KUKA KRL program: EPS_2_26115_SA7003_A_20260219035539.src

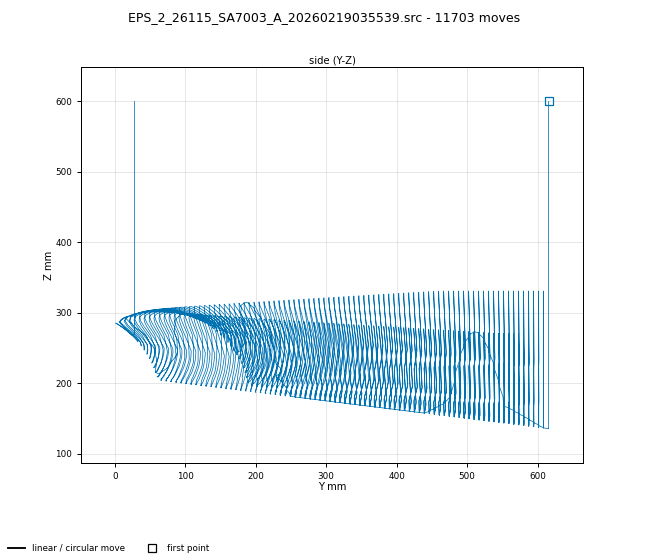
[picture p0: tool path of EPS_2_26115_SA7003_A_20260219035539.src, 11703 of 11705 moves have a stored position in this frame; points joined in program order, loops and branches not executed]
&ACCESS RVP
&REL 4
&COMMENT QRS 19112012
&PARAM EDITMASK = *
DEF PART()
EXT BAS (BAS_COMMAND :IN,REAL :IN )
INT I
BAS (#INITMOV,0 )

;KUKA QRS Post kuka4.cps  Date:22-06-2017 !

File_ID=3058

QRS_PRE_INIT()

;Init var - Until changes are made in qrs_pre_init
Outlet_Square_prg=0
Inlet_1_Square_prg=0
Inlet_2_Square_prg=0
Inlet_3_Square_prg=0
Inlet_4_Square_prg=0
Inlet_5_Square_prg=0

Outlet_1={X 0.000, Y 460.000, Z 230.500, B 0.000, E1 0.000 }
Inlet_1={X 0.000, Y 541.720, Z 170.500, B 0.000, E1 135.000 }
Outlet_1_type=201
Inlet_1_type=201
;QRS#1=Sidecore dimensions
;QRS#2=200-8" PVC SDR 35 Cut Back
;QRS#3=200-8" PVC SDR 35
;QRS#4=
;QRS#5=
;QRS#6=
;QRS#7=
;QRS#8=
;QRS#9=12-08 PSX
;QRS#10=12-08 PSX
;QRS#11=
;QRS#12=
;QRS#13=
;QRS#14=
;QRS#15=
;QRS#16=1220x127x610 2'
;QRS#17=EPS Height
;QRS#18=331
;QRS#19=*
;QRS#20= UPDATED VERSION 22-06-2017
;QRS#21=*
Outlet_Square=0100
Inlet_1_Square=0100
Inlet_2_Square=0
Inlet_3_Square=0
Inlet_4_Square=0
Inlet_5_Square=0
Mill_Square=1
Outlet_Square_Prg=214
Inlet_1_Square_prg=204

QRS_INIT()

$ADVANCE=5

; T1
PTP {E1 173.612,E2 173.612}
PTP {X 0,Y 615.504,A -85,B 0,C 180,E1 173.612,E2 173.612,E3 0,E4 0,E5 0,E6 0}
QRS_SPEED_INIT()
LIN {X 0,Y 615.504,Z 600,A -85,B 0,C 180,E1 173.612,E2 173.612,E3 0,E4 0,E5 0,E6 0} C_VEL
LIN {X 0,Y 615.504,Z 145.874,A -85,B 0,C 180,E1 173.612,E2 173.612} C_VEL
LIN {X 0,Y 615.504,Z 137.7,A -85,B 0,C 180,E1 173.612,E2 173.612} C_VEL
LIN {X 0,Y 615.487,Z 135.7,A -85,B 0,C 180,E1 173.425,E2 173.425} C_VEL
LIN {X 0,Y 615.477,Z 135.7,A -85,B 0,C 180,E1 170.801,E2 170.801} C_VEL
LIN {X 0,Y 615.494,Z 136.005,A -85,B 0,C 180,E1 170.138,E2 170.138} C_VEL
LIN {X 0,Y 615.486,Z 139.365,A -85,B 0,C 180,E1 167.47,E2 167.47} C_VEL
LIN {X 0,Y 615.476,Z 142.627,A -85,B 0,C 180,E1 164.774,E2 164.774} C_VEL
LIN {X 0,Y 615.48,Z 145.054,A -85,B 0,C 180,E1 162.73,E2 162.73} C_VEL
LIN {X 0,Y 615.448,Z 148.65,A -85,B 0,C 180,E1 159.966,E2 159.966} C_VEL
LIN {X 0,Y 615.448,Z 151.726,A -85,B 0,C 180,E1 157.664,E2 157.664} C_VEL
LIN {X 0,Y 615.492,Z 155.32,A -85,B 0,C 180,E1 155.009,E2 155.009} C_VEL
LIN {X 0,Y 615.478,Z 159.371,A -85,B 0,C 180,E1 152.085,E2 152.085} C_VEL
LIN {X 0,Y 615.499,Z 162.507,A -85,B 0,C 180,E1 149.841,E2 149.841} C_VEL
LIN {X 0,Y 615.459,Z 165.766,A -85,B 0,C 180,E1 147.541,E2 147.541} C_VEL
LIN {X 0,Y 615.495,Z 167.197,A -85,B 0,C 180,E1 146.54,E2 146.54} C_VEL
LIN {X 0,Y 615.491,Z 181.195,A -85,B 0,C 180,E1 146.222,E2 146.222} C_VEL
LIN {X 0,Y 615.454,Z 193.523,A -85,B 0,C 180,E1 145.809,E2 145.809} C_VEL
LIN {X 0,Y 615.455,Z 205.838,A -85,B 0,C 180,E1 145.244,E2 145.244} C_VEL
LIN {X 0,Y 615.495,Z 216.991,A -85,B 0,C 180,E1 144.586,E2 144.586} C_VEL
LIN {X 0,Y 615.5,Z 226.768,A -85,B 0,C 180,E1 143.872,E2 143.872} C_VEL
LIN {X 0,Y 615.497,Z 235.818,A -85,B 0,C 180,E1 143.063,E2 143.063} C_VEL
LIN {X 0,Y 615.494,Z 243.879,A -85,B 0,C 180,E1 142.181,E2 142.181} C_VEL
LIN {X 0,Y 615.493,Z 251.897,A -85,B 0,C 180,E1 141.097,E2 141.097} C_VEL
LIN {X 0,Y 615.498,Z 256.903,A -85,B 0,C 180,E1 140.251,E2 140.251} C_VEL
LIN {X 0,Y 615.498,Z 262.112,A -85,B 0,C 180,E1 139.15,E2 139.15} C_VEL
LIN {X 0,Y 615.498,Z 266.306,A -85,B 0,C 180,E1 137.919,E2 137.919} C_VEL
LIN {X 0,Y 615.496,Z 268.876,A -85,B 0,C 180,E1 136.757,E2 136.757} C_VEL
LIN {X 0,Y 615.495,Z 270.003,A -85,B 0,C 180,E1 135.852,E2 135.852} C_VEL
LIN {X 0,Y 615.496,Z 270.387,A -85,B 0,C 180,E1 134.933,E2 134.933} C_VEL
LIN {X 0,Y 615.493,Z 269.961,A -85,B 0,C 180,E1 133.999,E2 133.999} C_VEL
LIN {X 0,Y 615.496,Z 268.703,A -85,B 0,C 180,E1 133.049,E2 133.049} C_VEL
LIN {X 0,Y 615.495,Z 266.55,A -85,B 0,C 180,E1 132.082,E2 132.082} C_VEL
LIN {X 0,Y 615.494,Z 263.4,A -85,B 0,C 180,E1 131.096,E2 131.096} C_VEL
LIN {X 0,Y 615.497,Z 259.108,A -85,B 0,C 180,E1 130.091,E2 130.091} C_VEL
LIN {X 0,Y 615.498,Z 253.468,A -85,B 0,C 180,E1 129.064,E2 129.064} C_VEL
LIN {X 0,Y 615.495,Z 246.196,A -85,B 0,C 180,E1 128.014,E2 128.014} C_VEL
LIN {X 0,Y 615.497,Z 238.191,A -85,B 0,C 180,E1 127.09,E2 127.09} C_VEL
LIN {X 0,Y 615.499,Z 229.604,A -85,B 0,C 180,E1 126.277,E2 126.277} C_VEL
LIN {X 0,Y 615.494,Z 219.814,A -85,B 0,C 180,E1 125.515,E2 125.515} C_VEL
LIN {X 0,Y 615.456,Z 208.685,A -85,B 0,C 180,E1 124.817,E2 124.817} C_VEL
LIN {X 0,Y 615.443,Z 197.705,A -85,B 0,C 180,E1 124.276,E2 124.276} C_VEL
LIN {X 0,Y 615.472,Z 186.221,A -85,B 0,C 180,E1 123.841,E2 123.841} C_VEL
LIN {X 0,Y 615.497,Z 173.65,A -85,B 0,C 180,E1 123.498,E2 123.498} C_VEL
LIN {X 0,Y 615.498,Z 167.193,A -85,B 0,C 180,E1 123.367,E2 123.367} C_VEL
LIN {X 0,Y 615.469,Z 163.712,A -85,B 0,C 180,E1 120.921,E2 120.921} C_VEL
LIN {X 0,Y 615.485,Z 160.236,A -85,B 0,C 180,E1 118.451,E2 118.451} C_VEL
LIN {X 0,Y 615.485,Z 156.237,A -85,B 0,C 180,E1 115.569,E2 115.569} C_VEL
LIN {X 0,Y 615.482,Z 152.529,A -85,B 0,C 180,E1 112.845,E2 112.845} C_VEL
LIN {X 0,Y 615.445,Z 149.456,A -85,B 0,C 180,E1 110.548,E2 110.548} C_VEL
LIN {X 0,Y 615.454,Z 146.046,A -85,B 0,C 180,E1 107.958,E2 107.958} C_VEL
LIN {X 0,Y 615.495,Z 143.494,A -85,B 0,C 180,E1 105.905,E2 105.905} C_VEL
LIN {X 0,Y 615.485,Z 140.188,A -85,B 0,C 180,E1 103.201,E2 103.201} C_VEL
LIN {X 0,Y 615.487,Z 136.889,A -85,B 0,C 180,E1 100.527,E2 100.527} C_VEL
LIN {X 0,Y 615.494,Z 136.061,A -85,B 0,C 180,E1 99.862,E2 99.862} C_VEL
LIN {X 0,Y 615.487,Z 135.702,A -85,B 0,C 180,E1 98.537,E2 98.537} C_VEL
LIN {X 0,Y 615.499,Z 135.696,A -85,B 0,C 180,E1 95.899,E2 95.899} C_VEL
LIN {X 0,Y 615.47,Z 135.7,A -85,B 0,C 180,E1 93.273,E2 93.273} C_VEL
LIN {X 0,Y 615.466,Z 135.7,A -85,B 0,C 180,E1 90.654,E2 90.654} C_VEL
LIN {X 0,Y 615.5,Z 135.693,A -85,B 0,C 180,E1 88.037,E2 88.037} C_VEL
LIN {X 0,Y 615.487,Z 135.699,A -85,B 0,C 180,E1 85.416,E2 85.416} C_VEL
LIN {X 0,Y 615.489,Z 135.702,A -85,B 0,C 180,E1 82.784,E2 82.784} C_VEL
LIN {X 0,Y 615.493,Z 135.697,A -85,B 0,C 180,E1 80.138,E2 80.138} C_VEL
LIN {X 0,Y 615.464,Z 135.701,A -85,B 0,C 180,E1 77.469,E2 77.469} C_VEL
LIN {X 0,Y 615.469,Z 135.7,A -85,B 0,C 180,E1 74.774,E2 74.774} C_VEL
LIN {X 0,Y 615.494,Z 135.699,A -85,B 0,C 180,E1 72.043,E2 72.043} C_VEL
LIN {X 0,Y 615.481,Z 135.699,A -85,B 0,C 180,E1 69.269,E2 69.269} C_VEL
LIN {X 0,Y 615.49,Z 135.695,A -85,B 0,C 180,E1 66.444,E2 66.444} C_VEL
LIN {X 0,Y 615.487,Z 135.701,A -85,B 0,C 180,E1 63.556,E2 63.556} C_VEL
LIN {X 0,Y 615.492,Z 135.695,A -85,B 0,C 180,E1 60.594,E2 60.594} C_VEL
LIN {X 0,Y 615.477,Z 135.7,A -85,B 0,C 180,E1 57.67,E2 57.67} C_VEL
LIN {X 0,Y 615.484,Z 135.7,A -85,B 0,C 180,E1 55.185,E2 55.185} C_VEL
LIN {X 0,Y 615.497,Z 135.697,A -85,B 0,C 180,E1 52.759,E2 52.759} C_VEL
LIN {X 0,Y 615.476,Z 135.7,A -85,B 0,C 180,E1 49.912,E2 49.912} C_VEL
LIN {X 0,Y 615.491,Z 135.695,A -85,B 0,C 180,E1 46.952,E2 46.952} C_VEL
LIN {X 0,Y 615.494,Z 135.701,A -85,B 0,C 180,E1 44.148,E2 44.148} C_VEL
LIN {X 0,Y 615.491,Z 135.694,A -85,B 0,C 180,E1 41.095,E2 41.095} C_VEL
LIN {X 0,Y 615.491,Z 135.701,A -85,B 0,C 180,E1 38.068,E2 38.068} C_VEL
LIN {X 0,Y 615.496,Z 135.699,A -85,B 0,C 180,E1 35.615,E2 35.615} C_VEL
LIN {X 0,Y 615.487,Z 135.702,A -85,B 0,C 180,E1 33.236,E2 33.236} C_VEL
LIN {X 0,Y 615.496,Z 135.7,A -85,B 0,C 180,E1 30.919,E2 30.919} C_VEL
LIN {X 0,Y 615.495,Z 135.701,A -85,B 0,C 180,E1 28.451,E2 28.451} C_VEL
LIN {X 0,Y 615.49,Z 135.695,A -85,B 0,C 180,E1 25.569,E2 25.569} C_VEL
LIN {X 0,Y 615.475,Z 135.699,A -85,B 0,C 180,E1 22.845,E2 22.845} C_VEL
LIN {X 0,Y 615.467,Z 135.7,A -85,B 0,C 180,E1 20.551,E2 20.551} C_VEL
LIN {X 0,Y 615.472,Z 135.7,A -85,B 0,C 180,E1 17.957,E2 17.957} C_VEL
LIN {X 0,Y 615.494,Z 135.7,A -85,B 0,C 180,E1 15.225,E2 15.225} C_VEL
LIN {X 0,Y 615.482,Z 135.699,A -85,B 0,C 180,E1 12.53,E2 12.53} C_VEL
LIN {X 0,Y 615.496,Z 135.693,A -85,B 0,C 180,E1 9.862,E2 9.862} C_VEL
LIN {X 0,Y 615.473,Z 135.699,A -85,B 0,C 180,E1 7.215,E2 7.215} C_VEL
LIN {X 0,Y 615.477,Z 135.7,A -85,B 0,C 180,E1 4.584,E2 4.584} C_VEL
LIN {X 0,Y 615.5,Z 135.699,A -85,B 0,C 180,E1 1.963,E2 1.963} C_VEL
LIN {X 0,Y 615.483,Z 135.701,A -85,B 0,C 180,E1 -0.655,E2 -0.655} C_VEL
LIN {X 0,Y 615.479,Z 135.698,A -85,B 0,C 180,E1 -3.273,E2 -3.273} C_VEL
LIN {X 0,Y 615.498,Z 135.693,A -85,B 0,C 180,E1 -5.899,E2 -5.899} C_VEL
LIN {X 0,Y 615.472,Z 135.699,A -85,B 0,C 180,E1 -8.537,E2 -8.537} C_VEL
LIN {X 0,Y 615.482,Z 135.7,A -85,B 0,C 180,E1 -11.194,E2 -11.194} C_VEL
LIN {X 0,Y 615.486,Z 135.7,A -85,B 0,C 180,E1 -13.932,E2 -13.932} C_VEL
LIN {X 0,Y 615.471,Z 135.7,A -85,B 0,C 180,E1 -16.587,E2 -16.587} C_VEL
LIN {X 0,Y 615.485,Z 135.696,A -85,B 0,C 180,E1 -19.338,E2 -19.338} C_VEL
LIN {X 0,Y 615.49,Z 135.7,A -85,B 0,C 180,E1 -22.137,E2 -22.137} C_VEL
LIN {X 0,Y 615.486,Z 135.697,A -85,B 0,C 180,E1 -24.992,E2 -24.992} C_VEL
LIN {X 0,Y 615.482,Z 135.698,A -85,B 0,C 180,E1 -27.916,E2 -27.916} C_VEL
LIN {X 0,Y 615.465,Z 135.7,A -85,B 0,C 180,E1 -30.162,E2 -30.162} C_VEL
LIN {X 0,Y 615.466,Z 135.7,A -85,B 0,C 180,E1 -32.459,E2 -32.459} C_VEL
LIN {X 0,Y 615.481,Z 135.697,A -85,B 0,C 180,E1 -34.816,E2 -34.816} C_VEL
LIN {X 0,Y 615.494,Z 135.694,A -85,B 0,C 180,E1 -37.242,E2 -37.242} C_VEL
LIN {X 0,Y 615.475,Z 135.7,A -85,B 0,C 180,E1 -40.088,E2 -40.088} C_VEL
LIN {X 0,Y 615.467,Z 135.7,A -85,B 0,C 180,E1 -42.355,E2 -42.355} C_VEL
LIN {X 0,Y 615.497,Z 135.698,A -85,B 0,C 180,E1 -45.068,E2 -45.068} C_VEL
LIN {X 0,Y 615.474,Z 135.7,A -85,B 0,C 180,E1 -47.922,E2 -47.922} C_VEL
LIN {X 0,Y 615.498,Z 135.695,A -85,B 0,C 180,E1 -50.937,E2 -50.937} C_VEL
LIN {X 0,Y 615.487,Z 135.702,A -85,B 0,C 180,E1 -53.575,E2 -53.575} C_VEL
LIN {X 0,Y 615.475,Z 135.817,A -85,B 0,C 180,E1 -54.534,E2 -54.534} C_VEL
LIN {X 0,Y 615.449,Z 144.579,A -85,B 0,C 180,E1 -57.152,E2 -57.152} C_VEL
LIN {X 0,Y 615.438,Z 152.512,A -85,B 0,C 180,E1 -59.458,E2 -59.458} C_VEL
LIN {X 0,Y 615.482,Z 161.755,A -85,B 0,C 180,E1 -62.085,E2 -62.085} C_VEL
LIN {X 0,Y 615.484,Z 171.265,A -85,B 0,C 180,E1 -64.72,E2 -64.72} C_VEL
LIN {X 0,Y 615.471,Z 180.237,A -85,B 0,C 180,E1 -67.155,E2 -67.155} C_VEL
LIN {X 0,Y 615.489,Z 188.8,A -85,B 0,C 180,E1 -69.443,E2 -69.443} C_VEL
LIN {X 0,Y 615.499,Z 200.013,A -85,B 0,C 180,E1 -72.387,E2 -72.387} C_VEL
LIN {X 0,Y 615.48,Z 210.542,A -85,B 0,C 180,E1 -75.113,E2 -75.113} C_VEL
LIN {X 0,Y 615.455,Z 221.087,A -85,B 0,C 180,E1 -77.804,E2 -77.804} C_VEL
LIN {X 0,Y 615.498,Z 223.208,A -85,B 0,C 180,E1 -78.348,E2 -78.348} C_VEL
LIN {X 0,Y 615.497,Z 237.824,A -85,B 0,C 180,E1 -78.64,E2 -78.64} C_VEL
LIN {X 0,Y 615.453,Z 250.972,A -85,B 0,C 180,E1 -79.051,E2 -79.051} C_VEL
LIN {X 0,Y 615.442,Z 262.775,A -85,B 0,C 180,E1 -79.556,E2 -79.556} C_VEL
LIN {X 0,Y 615.489,Z 273.389,A -85,B 0,C 180,E1 -80.138,E2 -80.138} C_VEL
LIN {X 0,Y 615.498,Z 284.233,A -85,B 0,C 180,E1 -80.884,E2 -80.884} C_VEL
LIN {X 0,Y 615.497,Z 294.812,A -85,B 0,C 180,E1 -81.794,E2 -81.794} C_VEL
LIN {X 0,Y 615.498,Z 302.607,A -85,B 0,C 180,E1 -82.62,E2 -82.62} C_VEL
LIN {X 0,Y 615.496,Z 310.203,A -85,B 0,C 180,E1 -83.608,E2 -83.608} C_VEL
LIN {X 0,Y 615.498,Z 317.205,A -85,B 0,C 180,E1 -84.759,E2 -84.759} C_VEL
LIN {X 0,Y 615.494,Z 321.852,A -85,B 0,C 180,E1 -85.744,E2 -85.744} C_VEL
LIN {X 0,Y 615.494,Z 325.399,A -85,B 0,C 180,E1 -86.727,E2 -86.727} C_VEL
LIN {X 0,Y 615.497,Z 327.233,A -85,B 0,C 180,E1 -87.382,E2 -87.382} C_VEL
LIN {X 0,Y 615.5,Z 328.608,A -85,B 0,C 180,E1 -88.037,E2 -88.037} C_VEL
LIN {X 0,Y 615.496,Z 330.174,A -85,B 0,C 180,E1 -89.346,E2 -89.346} C_VEL
LIN {X 0,Y 615.494,Z 330.389,A -85,B 0,C 180,E1 -90,E2 -90} C_VEL
LIN {X 0,Y 615.495,Z 329.58,A -85,B 0,C 180,E1 -91.309,E2 -91.309} C_VEL
LIN {X 0,Y 615.5,Z 328.607,A -85,B 0,C 180,E1 -91.963,E2 -91.963} C_VEL
LIN {X 0,Y 615.497,Z 327.233,A -85,B 0,C 180,E1 -92.618,E2 -92.618} C_VEL
LIN {X 0,Y 615.496,Z 324.349,A -85,B 0,C 180,E1 -93.601,E2 -93.601} C_VEL
LIN {X 0,Y 615.498,Z 320.441,A -85,B 0,C 180,E1 -94.585,E2 -94.585} C_VEL
LIN {X 0,Y 615.499,Z 315.404,A -85,B 0,C 180,E1 -95.57,E2 -95.57} C_VEL
LIN {X 0,Y 615.497,Z 308.87,A -85,B 0,C 180,E1 -96.583,E2 -96.583} C_VEL
LIN {X 0,Y 615.497,Z 301.132,A -85,B 0,C 180,E1 -97.546,E2 -97.546} C_VEL
LIN {X 0,Y 615.498,Z 293.043,A -85,B 0,C 180,E1 -98.371,E2 -98.371} C_VEL
LIN {X 0,Y 615.499,Z 283.165,A -85,B 0,C 180,E1 -99.199,E2 -99.199} C_VEL
LIN {X 0,Y 615.479,Z 271.98,A -85,B 0,C 180,E1 -99.945,E2 -99.945} C_VEL
LIN {X 0,Y 615.441,Z 261.027,A -85,B 0,C 180,E1 -100.528,E2 -100.528} C_VEL
LIN {X 0,Y 615.459,Z 248.774,A -85,B 0,C 180,E1 -101.031,E2 -101.031} C_VEL
LIN {X 0,Y 615.499,Z 236.056,A -85,B 0,C 180,E1 -101.402,E2 -101.402} C_VEL
LIN {X 0,Y 615.498,Z 223.208,A -85,B 0,C 180,E1 -101.652,E2 -101.652} C_VEL
LIN {X 0,Y 615.46,Z 213.08,A -85,B 0,C 180,E1 -104.239,E2 -104.239} C_VEL
LIN {X 0,Y 615.491,Z 202.639,A -85,B 0,C 180,E1 -106.928,E2 -106.928} C_VEL
LIN {X 0,Y 615.487,Z 192.103,A -85,B 0,C 180,E1 -109.685,E2 -109.685} C_VEL
LIN {X 0,Y 615.491,Z 182.087,A -85,B 0,C 180,E1 -112.346,E2 -112.346} C_VEL
LIN {X 0,Y 615.467,Z 172.322,A -85,B 0,C 180,E1 -114.993,E2 -114.993} C_VEL
LIN {X 0,Y 615.496,Z 163.073,A -85,B 0,C 180,E1 -117.545,E2 -117.545} C_VEL
LIN {X 0,Y 615.448,Z 153.832,A -85,B 0,C 180,E1 -120.162,E2 -120.162} C_VEL
LIN {X 0,Y 615.429,Z 145.902,A -85,B 0,C 180,E1 -122.461,E2 -122.461} C_VEL
LIN {X 0,Y 615.496,Z 136.642,A -85,B 0,C 180,E1 -125.214,E2 -125.214} C_VEL
LIN {X 0,Y 615.479,Z 135.7,A -85,B 0,C 180,E1 -125.516,E2 -125.516} C_VEL
LIN {X 0,Y 615.49,Z 135.7,A -85,B 0,C 180,E1 -128.069,E2 -128.069} C_VEL
LIN {X 0,Y 615.49,Z 135.7,A -85,B 0,C 180,E1 -131.094,E2 -131.094} C_VEL
LIN {X 0,Y 615.483,Z 135.7,A -85,B 0,C 180,E1 -133.997,E2 -133.997} C_VEL
LIN {X 0,Y 615.488,Z 135.697,A -85,B 0,C 180,E1 -136.755,E2 -136.755} C_VEL
LIN {X 0,Y 615.485,Z 135.701,A -85,B 0,C 180,E1 -139.393,E2 -139.393} C_VEL
LIN {X 0,Y 615.477,Z 135.701,A -85,B 0,C 180,E1 -141.99,E2 -141.99} C_VEL
LIN {X 0,Y 615.498,Z 135.699,A -85,B 0,C 180,E1 -144.385,E2 -144.385} C_VEL
LIN {X 0,Y 615.492,Z 135.697,A -85,B 0,C 180,E1 -146.764,E2 -146.764} C_VEL
LIN {X 0,Y 615.489,Z 135.698,A -85,B 0,C 180,E1 -149.08,E2 -149.08} C_VEL
LIN {X 0,Y 615.486,Z 135.7,A -85,B 0,C 180,E1 -151.551,E2 -151.551} C_VEL
LIN {X 0,Y 615.499,Z 135.7,A -85,B 0,C 180,E1 -154.43,E2 -154.43} C_VEL
LIN {X 0,Y 615.482,Z 135.7,A -85,B 0,C 180,E1 -157.155,E2 -157.155} C_VEL
LIN {X 0,Y 615.476,Z 135.7,A -85,B 0,C 180,E1 -159.967,E2 -159.967} C_VEL
LIN {X 0,Y 615.484,Z 135.7,A -85,B 0,C 180,E1 -162.729,E2 -162.729} C_VEL
LIN {X 0,Y 615.493,Z 135.7,A -85,B 0,C 180,E1 -165.451,E2 -165.451} C_VEL
LIN {X 0,Y 615.49,Z 135.697,A -85,B 0,C 180,E1 -168.139,E2 -168.139} C_VEL
LIN {X 0,Y 615.484,Z 135.7,A -85,B 0,C 180,E1 -170.801,E2 -170.801} C_VEL
LIN {X 0,Y 615.487,Z 135.7,A -85,B 0,C 180,E1 -173.443,E2 -173.443} C_VEL
LIN {X 0,Y 615.493,Z 135.696,A -85,B 0,C 180,E1 -176.071,E2 -176.071} C_VEL
LIN {X 0,Y 615.495,Z 135.7,A -85,B 0,C 180,E1 -178.691,E2 -178.691} C_VEL
LIN {X 0,Y 615.478,Z 135.7,A -85,B 0,C 180,E1 -181.308,E2 -181.308} C_VEL
LIN {X 0,Y 615.492,Z 135.698,A -85,B 0,C 180,E1 -183.928,E2 -183.928} C_VEL
LIN {X 0,Y 615.487,Z 135.7,A -85,B 0,C 180,E1 -186.575,E2 -186.575} C_VEL
LIN {X 0,Y 614.798,Z 135.845,A -85,B 0,C 180,E1 -187.121,E2 -187.121} C_VEL
LIN {X 0,Y 611.938,Z 136.262,A -85,B 0,C 180,E1 -188.007,E2 -188.007} C_VEL
LIN {X 0,Y 609.539,Z 136.563,A -85,B 0,C 180,E1 -188.719,E2 -188.719} C_VEL
LIN {X 0,Y 608.516,Z 136.702,A -85,B 0,C 180,E1 -189.269,E2 -189.269} C_VEL
LIN {X 0,Y 608.436,Z 136.768,A -85,B 0,C 180,E1 -189.455,E2 -189.455} C_VEL
LIN {X 0,Y 608.462,Z 137.016,A -85,B 0,C 180,E1 -189.977,E2 -189.977} C_VEL
LIN {X 0,Y 608.45,Z 140.401,A -85,B 0,C 180,E1 -192.677,E2 -192.677} C_VEL
LIN {X 0,Y 608.442,Z 143.694,A -85,B 0,C 180,E1 -195.406,E2 -195.406} C_VEL
LIN {X 0,Y 608.442,Z 146.154,A -85,B 0,C 180,E1 -197.476,E2 -197.476} C_VEL
LIN {X 0,Y 608.387,Z 149.724,A -85,B 0,C 180,E1 -200.276,E2 -200.276} C_VEL
LIN {X 0,Y 608.407,Z 153.52,A -85,B 0,C 180,E1 -203.125,E2 -203.125} C_VEL
LIN {X 0,Y 608.413,Z 157.48,A -85,B 0,C 180,E1 -206.037,E2 -206.037} C_VEL
LIN {X 0,Y 608.418,Z 161.039,A -85,B 0,C 180,E1 -208.61,E2 -208.61} C_VEL
LIN {X 0,Y 608.417,Z 164.837,A -85,B 0,C 180,E1 -211.319,E2 -211.319} C_VEL
LIN {X 0,Y 608.427,Z 167.679,A -85,B 0,C 180,E1 -213.325,E2 -213.325} C_VEL
LIN {X 0,Y 608.523,Z 182.01,A -85,B 0,C 180,E1 -213.667,E2 -213.667} C_VEL
LIN {X 0,Y 608.478,Z 193.76,A -85,B 0,C 180,E1 -214.069,E2 -214.069} C_VEL
LIN {X 0,Y 608.455,Z 206.067,A -85,B 0,C 180,E1 -214.64,E2 -214.64} C_VEL
LIN {X 0,Y 608.494,Z 216.768,A -85,B 0,C 180,E1 -215.274,E2 -215.274} C_VEL
LIN {X 0,Y 608.486,Z 227.821,A -85,B 0,C 180,E1 -216.089,E2 -216.089} C_VEL
LIN {X 0,Y 608.46,Z 238.007,A -85,B 0,C 180,E1 -217.036,E2 -217.036} C_VEL
LIN {X 0,Y 608.453,Z 246.33,A -85,B 0,C 180,E1 -217.991,E2 -217.991} C_VEL
LIN {X 0,Y 608.437,Z 254.12,A -85,B 0,C 180,E1 -219.12,E2 -219.12} C_VEL
LIN {X 0,Y 608.452,Z 260.471,A -85,B 0,C 180,E1 -220.303,E2 -220.303} C_VEL
LIN {X 0,Y 608.427,Z 264.671,A -85,B 0,C 180,E1 -221.338,E2 -221.338} C_VEL
LIN {X 0,Y 608.438,Z 267.636,A -85,B 0,C 180,E1 -222.331,E2 -222.331} C_VEL
LIN {X 0,Y 608.433,Z 269.609,A -85,B 0,C 180,E1 -223.305,E2 -223.305} C_VEL
LIN {X 0,Y 608.418,Z 270.697,A -85,B 0,C 180,E1 -224.26,E2 -224.26} C_VEL
LIN {X 0,Y 608.417,Z 270.97,A -85,B 0,C 180,E1 -225.2,E2 -225.2} C_VEL
LIN {X 0,Y 608.427,Z 270.469,A -85,B 0,C 180,E1 -226.126,E2 -226.126} C_VEL
LIN {X 0,Y 608.435,Z 269.189,A -85,B 0,C 180,E1 -227.038,E2 -227.038} C_VEL
LIN {X 0,Y 608.425,Z 267.164,A -85,B 0,C 180,E1 -227.935,E2 -227.935} C_VEL
LIN {X 0,Y 608.431,Z 264.414,A -85,B 0,C 180,E1 -228.821,E2 -228.821} C_VEL
LIN {X 0,Y 608.444,Z 259.863,A -85,B 0,C 180,E1 -229.912,E2 -229.912} C_VEL
LIN {X 0,Y 608.438,Z 253.597,A -85,B 0,C 180,E1 -231.056,E2 -231.056} C_VEL
LIN {X 0,Y 608.453,Z 247.02,A -85,B 0,C 180,E1 -232.008,E2 -232.008} C_VEL
LIN {X 0,Y 608.459,Z 238.894,A -85,B 0,C 180,E1 -232.963,E2 -232.963} C_VEL
LIN {X 0,Y 608.483,Z 228.88,A -85,B 0,C 180,E1 -233.91,E2 -233.91} C_VEL
LIN {X 0,Y 608.486,Z 218.16,A -85,B 0,C 180,E1 -234.725,E2 -234.725} C_VEL
LIN {X 0,Y 608.452,Z 206.176,A -85,B 0,C 180,E1 -235.444,E2 -235.444} C_VEL
LIN {X 0,Y 608.478,Z 194.728,A -85,B 0,C 180,E1 -235.981,E2 -235.981} C_VEL
LIN {X 0,Y 608.523,Z 181.703,A -85,B 0,C 180,E1 -236.432,E2 -236.432} C_VEL
LIN {X 0,Y 608.444,Z 167.665,A -85,B 0,C 180,E1 -236.774,E2 -236.774} C_VEL
LIN {X 0,Y 608.415,Z 163.878,A -85,B 0,C 180,E1 -239.452,E2 -239.452} C_VEL
LIN {X 0,Y 608.43,Z 160.688,A -85,B 0,C 180,E1 -241.732,E2 -241.732} C_VEL
LIN {X 0,Y 608.43,Z 156.596,A -85,B 0,C 180,E1 -244.698,E2 -244.698} C_VEL
LIN {X 0,Y 608.411,Z 152.677,A -85,B 0,C 180,E1 -247.592,E2 -247.592} C_VEL
LIN {X 0,Y 608.42,Z 148.913,A -85,B 0,C 180,E1 -250.428,E2 -250.428} C_VEL
LIN {X 0,Y 608.435,Z 145.048,A -85,B 0,C 180,E1 -253.48,E2 -253.48} C_VEL
LIN {X 0,Y 608.436,Z 142.005,A -85,B 0,C 180,E1 -255.994,E2 -255.994} C_VEL
LIN {X 0,Y 608.451,Z 138.705,A -85,B 0,C 180,E1 -258.676,E2 -258.676} C_VEL
LIN {X 0,Y 608.462,Z 137.049,A -85,B 0,C 180,E1 -260.023,E2 -260.023} C_VEL
LIN {X 0,Y 608.454,Z 136.697,A -85,B 0,C 180,E1 -261.364,E2 -261.364} C_VEL
LIN {X 0,Y 608.491,Z 136.692,A -85,B 0,C 180,E1 -264.033,E2 -264.033} C_VEL
LIN {X 0,Y 608.466,Z 136.693,A -85,B 0,C 180,E1 -266.689,E2 -266.689} C_VEL
LIN {X 0,Y 608.462,Z 136.693,A -85,B 0,C 180,E1 -269.338,E2 -269.338} C_VEL
LIN {X 0,Y 608.469,Z 136.693,A -85,B 0,C 180,E1 -271.986,E2 -271.986} C_VEL
LIN {X 0,Y 608.454,Z 136.696,A -85,B 0,C 180,E1 -274.638,E2 -274.638} C_VEL
LIN {X 0,Y 608.466,Z 136.696,A -85,B 0,C 180,E1 -277.299,E2 -277.299} C_VEL
LIN {X 0,Y 608.46,Z 136.694,A -85,B 0,C 180,E1 -279.977,E2 -279.977} C_VEL
LIN {X 0,Y 608.461,Z 136.693,A -85,B 0,C 180,E1 -282.677,E2 -282.677} C_VEL
LIN {X 0,Y 608.457,Z 136.695,A -85,B 0,C 180,E1 -285.406,E2 -285.406} C_VEL
LIN {X 0,Y 608.447,Z 136.698,A -85,B 0,C 180,E1 -288.172,E2 -288.172} C_VEL
LIN {X 0,Y 608.455,Z 136.694,A -85,B 0,C 180,E1 -290.982,E2 -290.982} C_VEL
LIN {X 0,Y 608.473,Z 136.693,A -85,B 0,C 180,E1 -293.845,E2 -293.845} C_VEL
LIN {X 0,Y 608.447,Z 136.696,A -85,B 0,C 180,E1 -296.774,E2 -296.774} C_VEL
LIN {X 0,Y 608.469,Z 136.693,A -85,B 0,C 180,E1 -299.779,E2 -299.779} C_VEL
LIN {X 0,Y 608.459,Z 136.697,A -85,B 0,C 180,E1 -302.523,E2 -302.523} C_VEL
LIN {X 0,Y 608.436,Z 136.697,A -85,B 0,C 180,E1 -305.278,E2 -305.278} C_VEL
LIN {X 0,Y 608.46,Z 136.694,A -85,B 0,C 180,E1 -307.747,E2 -307.747} C_VEL
LIN {X 0,Y 608.438,Z 136.696,A -85,B 0,C 180,E1 -310.328,E2 -310.328} C_VEL
LIN {X 0,Y 608.458,Z 136.694,A -85,B 0,C 180,E1 -312.959,E2 -312.959} C_VEL
LIN {X 0,Y 608.463,Z 136.696,A -85,B 0,C 180,E1 -315.736,E2 -315.736} C_VEL
LIN {X 0,Y 608.466,Z 136.693,A -85,B 0,C 180,E1 -318.657,E2 -318.657} C_VEL
LIN {X 0,Y 608.469,Z 136.692,A -85,B 0,C 180,E1 -321.413,E2 -321.413} C_VEL
LIN {X 0,Y 608.444,Z 136.696,A -85,B 0,C 180,E1 -323.955,E2 -323.955} C_VEL
LIN {X 0,Y 608.442,Z 136.696,A -85,B 0,C 180,E1 -326.328,E2 -326.328} C_VEL
LIN {X 0,Y 608.48,Z 136.691,A -85,B 0,C 180,E1 -328.727,E2 -328.727} C_VEL
LIN {X 0,Y 608.475,Z 136.694,A -85,B 0,C 180,E1 -331.38,E2 -331.38} C_VEL
LIN {X 0,Y 608.474,Z 136.693,A -85,B 0,C 180,E1 -334.279,E2 -334.279} C_VEL
LIN {X 0,Y 608.446,Z 136.695,A -85,B 0,C 180,E1 -336.876,E2 -336.876} C_VEL
LIN {X 0,Y 608.452,Z 136.694,A -85,B 0,C 180,E1 -339.326,E2 -339.326} C_VEL
LIN {X 0,Y 608.437,Z 136.696,A -85,B 0,C 180,E1 -341.828,E2 -341.828} C_VEL
LIN {X 0,Y 608.477,Z 136.693,A -85,B 0,C 180,E1 -344.595,E2 -344.595} C_VEL
LIN {X 0,Y 608.471,Z 136.695,A -85,B 0,C 180,E1 -347.323,E2 -347.323} C_VEL
LIN {X 0,Y 608.464,Z 136.693,A -85,B 0,C 180,E1 -350.023,E2 -350.023} C_VEL
LIN {X 0,Y 608.441,Z 136.696,A -85,B 0,C 180,E1 -352.701,E2 -352.701} C_VEL
LIN {X 0,Y 608.445,Z 136.696,A -85,B 0,C 180,E1 -355.363,E2 -355.363} C_VEL
LIN {X 0,Y 608.468,Z 136.695,A -85,B 0,C 180,E1 -358.015,E2 -358.015} C_VEL
LIN {X 0,Y 608.477,Z 136.693,A -85,B 0,C 180,E1 -360.662,E2 -360.662} C_VEL
LIN {X 0,Y 608.474,Z 136.692,A -85,B 0,C 180,E1 -363.311,E2 -363.311} C_VEL
LIN {X 0,Y 608.471,Z 136.692,A -85,B 0,C 180,E1 -365.967,E2 -365.967} C_VEL
LIN {X 0,Y 608.446,Z 136.696,A -85,B 0,C 180,E1 -368.636,E2 -368.636} C_VEL
LIN {X 0,Y 608.476,Z 136.695,A -85,B 0,C 180,E1 -371.324,E2 -371.324} C_VEL
LIN {X 0,Y 608.472,Z 136.693,A -85,B 0,C 180,E1 -374.038,E2 -374.038} C_VEL
LIN {X 0,Y 608.439,Z 136.696,A -85,B 0,C 180,E1 -376.785,E2 -376.785} C_VEL
LIN {X 0,Y 608.45,Z 136.696,A -85,B 0,C 180,E1 -379.571,E2 -379.571} C_VEL
LIN {X 0,Y 608.462,Z 136.695,A -85,B 0,C 180,E1 -382.477,E2 -382.477} C_VEL
LIN {X 0,Y 608.454,Z 136.694,A -85,B 0,C 180,E1 -385.301,E2 -385.301} C_VEL
LIN {X 0,Y 608.454,Z 136.694,A -85,B 0,C 180,E1 -387.518,E2 -387.518} C_VEL
LIN {X 0,Y 608.436,Z 136.696,A -85,B 0,C 180,E1 -389.966,E2 -389.966} C_VEL
LIN {X 0,Y 608.446,Z 136.695,A -85,B 0,C 180,E1 -392.52,E2 -392.52} C_VEL
LIN {X 0,Y 608.444,Z 136.697,A -85,B 0,C 180,E1 -395.278,E2 -395.278} C_VEL
LIN {X 0,Y 608.47,Z 136.694,A -85,B 0,C 180,E1 -397.747,E2 -397.747} C_VEL
LIN {X 0,Y 608.447,Z 136.699,A -85,B 0,C 180,E1 -400.328,E2 -400.328} C_VEL
LIN {X 0,Y 608.475,Z 136.691,A -85,B 0,C 180,E1 -403.309,E2 -403.309} C_VEL
LIN {X 0,Y 608.46,Z 136.695,A -85,B 0,C 180,E1 -406.13,E2 -406.13} C_VEL
LIN {X 0,Y 608.454,Z 136.698,A -85,B 0,C 180,E1 -408.823,E2 -408.823} C_VEL
LIN {X 0,Y 608.44,Z 136.698,A -85,B 0,C 180,E1 -411.41,E2 -411.41} C_VEL
LIN {X 0,Y 608.444,Z 136.697,A -85,B 0,C 180,E1 -413.955,E2 -413.955} C_VEL
LIN {X 0,Y 608.468,Z 136.815,A -85,B 0,C 180,E1 -414.369,E2 -414.369} C_VEL
LIN {X 0,Y 608.499,Z 145.917,A -85,B 0,C 180,E1 -417.123,E2 -417.123} C_VEL
LIN {X 0,Y 608.468,Z 153.86,A -85,B 0,C 180,E1 -419.455,E2 -419.455} C_VEL
LIN {X 0,Y 608.495,Z 163.127,A -85,B 0,C 180,E1 -422.111,E2 -422.111} C_VEL
LIN {X 0,Y 608.475,Z 172.395,A -85,B 0,C 180,E1 -424.7,E2 -424.7} C_VEL
LIN {X 0,Y 608.48,Z 182.986,A -85,B 0,C 180,E1 -427.595,E2 -427.595} C_VEL
LIN {X 0,Y 608.459,Z 193.577,A -85,B 0,C 180,E1 -430.43,E2 -430.43} C_VEL
LIN {X 0,Y 608.45,Z 204.168,A -85,B 0,C 180,E1 -433.216,E2 -433.216} C_VEL
LIN {X 0,Y 608.439,Z 214.889,A -85,B 0,C 180,E1 -435.995,E2 -435.995} C_VEL
LIN {X 0,Y 608.438,Z 223.572,A -85,B 0,C 180,E1 -438.222,E2 -438.222} C_VEL
LIN {X 0,Y 608.55,Z 237.098,A -85,B 0,C 180,E1 -438.488,E2 -438.488} C_VEL
LIN {X 0,Y 608.487,Z 249.517,A -85,B 0,C 180,E1 -438.865,E2 -438.865} C_VEL
LIN {X 0,Y 608.467,Z 261.173,A -85,B 0,C 180,E1 -439.35,E2 -439.35} C_VEL
LIN {X 0,Y 608.478,Z 273.58,A -85,B 0,C 180,E1 -440.023,E2 -440.023} C_VEL
LIN {X 0,Y 608.483,Z 284.475,A -85,B 0,C 180,E1 -440.778,E2 -440.778} C_VEL
LIN {X 0,Y 608.475,Z 295.113,A -85,B 0,C 180,E1 -441.699,E2 -441.699} C_VEL
LIN {X 0,Y 608.471,Z 302.961,A -85,B 0,C 180,E1 -442.534,E2 -442.534} C_VEL
LIN {X 0,Y 608.461,Z 310.287,A -85,B 0,C 180,E1 -443.485,E2 -443.485} C_VEL
LIN {X 0,Y 608.451,Z 315.866,A -85,B 0,C 180,E1 -444.366,E2 -444.366} C_VEL
LIN {X 0,Y 608.432,Z 320.95,A -85,B 0,C 180,E1 -445.362,E2 -445.362} C_VEL
LIN {X 0,Y 608.449,Z 324.896,A -85,B 0,C 180,E1 -446.358,E2 -446.358} C_VEL
LIN {X 0,Y 608.425,Z 327.809,A -85,B 0,C 180,E1 -447.352,E2 -447.352} C_VEL
LIN {X 0,Y 608.445,Z 329.201,A -85,B 0,C 180,E1 -448.014,E2 -448.014} C_VEL
LIN {X 0,Y 608.438,Z 330.783,A -85,B 0,C 180,E1 -449.338,E2 -449.338} C_VEL
LIN {X 0,Y 608.434,Z 331,A -85,B 0,C 180,E1 -450,E2 -450} C_VEL
LIN {X 0,Y 608.448,Z 330.184,A -85,B 0,C 180,E1 -451.324,E2 -451.324} C_VEL
LIN {X 0,Y 608.445,Z 329.201,A -85,B 0,C 180,E1 -451.986,E2 -451.986} C_VEL
LIN {X 0,Y 608.425,Z 327.809,A -85,B 0,C 180,E1 -452.648,E2 -452.648} C_VEL
LIN {X 0,Y 608.449,Z 324.896,A -85,B 0,C 180,E1 -453.643,E2 -453.643} C_VEL
LIN {X 0,Y 608.432,Z 320.949,A -85,B 0,C 180,E1 -454.638,E2 -454.638} C_VEL
LIN {X 0,Y 608.438,Z 314.876,A -85,B 0,C 180,E1 -455.801,E2 -455.801} C_VEL
LIN {X 0,Y 608.462,Z 308.234,A -85,B 0,C 180,E1 -456.799,E2 -456.799} C_VEL
LIN {X 0,Y 608.456,Z 299.988,A -85,B 0,C 180,E1 -457.8,E2 -457.8} C_VEL
LIN {X 0,Y 608.472,Z 291.534,A -85,B 0,C 180,E1 -458.636,E2 -458.636} C_VEL
LIN {X 0,Y 608.48,Z 281.088,A -85,B 0,C 180,E1 -459.473,E2 -459.473} C_VEL
LIN {X 0,Y 608.488,Z 270.752,A -85,B 0,C 180,E1 -460.145,E2 -460.145} C_VEL
LIN {X 0,Y 608.466,Z 259.856,A -85,B 0,C 180,E1 -460.713,E2 -460.713} C_VEL
LIN {X 0,Y 608.493,Z 248.085,A -85,B 0,C 180,E1 -461.186,E2 -461.186} C_VEL
LIN {X 0,Y 608.551,Z 235.26,A -85,B 0,C 180,E1 -461.555,E2 -461.555} C_VEL
LIN {X 0,Y 608.442,Z 223.53,A -85,B 0,C 180,E1 -461.789,E2 -461.789} C_VEL
LIN {X 0,Y 608.41,Z 213.435,A -85,B 0,C 180,E1 -464.38,E2 -464.38} C_VEL
LIN {X 0,Y 608.45,Z 204.167,A -85,B 0,C 180,E1 -466.784,E2 -466.784} C_VEL
LIN {X 0,Y 608.46,Z 193.576,A -85,B 0,C 180,E1 -469.571,E2 -469.571} C_VEL
LIN {X 0,Y 608.463,Z 182.724,A -85,B 0,C 180,E1 -472.476,E2 -472.476} C_VEL
LIN {X 0,Y 608.475,Z 172.394,A -85,B 0,C 180,E1 -475.3,E2 -475.3} C_VEL
LIN {X 0,Y 608.495,Z 163.126,A -85,B 0,C 180,E1 -477.89,E2 -477.89} C_VEL
LIN {X 0,Y 608.469,Z 153.859,A -85,B 0,C 180,E1 -480.545,E2 -480.545} C_VEL
LIN {X 0,Y 608.52,Z 144.592,A -85,B 0,C 180,E1 -483.271,E2 -483.271} C_VEL
LIN {X 0,Y 608.471,Z 136.694,A -85,B 0,C 180,E1 -485.682,E2 -485.682} C_VEL
LIN {X 0,Y 608.471,Z 136.696,A -85,B 0,C 180,E1 -488.24,E2 -488.24} C_VEL
LIN {X 0,Y 608.462,Z 136.696,A -85,B 0,C 180,E1 -491.342,E2 -491.342} C_VEL
LIN {X 0,Y 608.462,Z 136.697,A -85,B 0,C 180,E1 -494.264,E2 -494.264} C_VEL
LIN {X 0,Y 608.457,Z 136.696,A -85,B 0,C 180,E1 -497.04,E2 -497.04} C_VEL
LIN {X 0,Y 608.457,Z 136.695,A -85,B 0,C 180,E1 -499.697,E2 -499.697} C_VEL
LIN {X 0,Y 608.467,Z 136.696,A -85,B 0,C 180,E1 -502.253,E2 -502.253} C_VEL
LIN {X 0,Y 608.485,Z 136.692,A -85,B 0,C 180,E1 -505.09,E2 -505.09} C_VEL
LIN {X 0,Y 608.465,Z 136.694,A -85,B 0,C 180,E1 -507.905,E2 -507.905} C_VEL
LIN {X 0,Y 608.47,Z 136.695,A -85,B 0,C 180,E1 -510.22,E2 -510.22} C_VEL
LIN {X 0,Y 608.481,Z 136.692,A -85,B 0,C 180,E1 -512.793,E2 -512.793} C_VEL
LIN {X 0,Y 608.45,Z 136.699,A -85,B 0,C 180,E1 -515.428,E2 -515.428} C_VEL
LIN {X 0,Y 608.47,Z 136.695,A -85,B 0,C 180,E1 -518.308,E2 -518.308} C_VEL
LIN {X 0,Y 608.476,Z 136.694,A -85,B 0,C 180,E1 -521.284,E2 -521.284} C_VEL
LIN {X 0,Y 608.462,Z 136.694,A -85,B 0,C 180,E1 -523.906,E2 -523.906} C_VEL
LIN {X 0,Y 608.462,Z 136.696,A -85,B 0,C 180,E1 -526.643,E2 -526.643} C_VEL
LIN {X 0,Y 608.465,Z 136.695,A -85,B 0,C 180,E1 -529.35,E2 -529.35} C_VEL
LIN {X 0,Y 608.483,Z 136.692,A -85,B 0,C 180,E1 -532.033,E2 -532.033} C_VEL
LIN {X 0,Y 608.469,Z 136.695,A -85,B 0,C 180,E1 -534.698,E2 -534.698} C_VEL
LIN {X 0,Y 608.474,Z 136.693,A -85,B 0,C 180,E1 -537.352,E2 -537.352} C_VEL
LIN {X 0,Y 608.484,Z 136.692,A -85,B 0,C 180,E1 -540,E2 -540} C_VEL
LIN {X 0,Y 608.481,Z 136.694,A -85,B 0,C 180,E1 -542.648,E2 -542.648} C_VEL
LIN {X 0,Y 608.457,Z 136.695,A -85,B 0,C 180,E1 -545.302,E2 -545.302} C_VEL
LIN {X 0,Y 608.481,Z 136.693,A -85,B 0,C 180,E1 -547.967,E2 -547.967} C_VEL
LIN {X 0,Y 608.436,Z 136.768,A -85,B 0,C 180,E1 -549.455,E2 -549.455} C_VEL
LIN {X 0,Y 607.772,Z 137.224,A -85,B 0,C 180,E1 -550.006,E2 -550.006} C_VEL
LIN {X 0,Y 604.904,Z 138.492,A -85,B 0,C 180,E1 -550.895,E2 -550.895} C_VEL
LIN {X 0,Y 602.477,Z 139.614,A -85,B 0,C 180,E1 -551.609,E2 -551.609} C_VEL
LIN {X 0,Y 601.436,Z 140.391,A -85,B 0,C 180,E1 -552.161,E2 -552.161} C_VEL
LIN {X 0,Y 601.353,Z 140.628,A -85,B 0,C 180,E1 -552.349,E2 -552.349} C_VEL
LIN {X 0,Y 601.369,Z 143.712,A -85,B 0,C 180,E1 -554.898,E2 -554.898} C_VEL
LIN {X 0,Y 601.374,Z 147.038,A -85,B 0,C 180,E1 -557.689,E2 -557.689} C_VEL
LIN {X 0,Y 601.329,Z 150.775,A -85,B 0,C 180,E1 -560.772,E2 -560.772} C_VEL
LIN {X 0,Y 601.326,Z 154.266,A -85,B 0,C 180,E1 -563.414,E2 -563.414} C_VEL
LIN {X 0,Y 601.325,Z 157.542,A -85,B 0,C 180,E1 -565.849,E2 -565.849} C_VEL
LIN {X 0,Y 601.327,Z 161.344,A -85,B 0,C 180,E1 -568.632,E2 -568.632} C_VEL
LIN {X 0,Y 601.317,Z 164.55,A -85,B 0,C 180,E1 -570.947,E2 -570.947} C_VEL
LIN {X 0,Y 601.337,Z 167.689,A -85,B 0,C 180,E1 -573.192,E2 -573.192} C_VEL
LIN {X 0,Y 601.608,Z 173.507,A -85,B 0,C 180,E1 -573.314,E2 -573.314} C_VEL
LIN {X 0,Y 601.559,Z 185.9,A -85,B 0,C 180,E1 -573.656,E2 -573.656} C_VEL
LIN {X 0,Y 601.473,Z 197.838,A -85,B 0,C 180,E1 -574.115,E2 -574.115} C_VEL
LIN {X 0,Y 601.475,Z 209.803,A -85,B 0,C 180,E1 -574.724,E2 -574.724} C_VEL
LIN {X 0,Y 601.466,Z 221.496,A -85,B 0,C 180,E1 -575.49,E2 -575.49} C_VEL
LIN {X 0,Y 601.439,Z 231.051,A -85,B 0,C 180,E1 -576.265,E2 -576.265} C_VEL
LIN {X 0,Y 601.415,Z 240.303,A -85,B 0,C 180,E1 -577.188,E2 -577.188} C_VEL
LIN {X 0,Y 601.391,Z 249.001,A -85,B 0,C 180,E1 -578.27,E2 -578.27} C_VEL
LIN {X 0,Y 601.384,Z 255.761,A -85,B 0,C 180,E1 -579.325,E2 -579.325} C_VEL
LIN {X 0,Y 601.336,Z 261.846,A -85,B 0,C 180,E1 -580.564,E2 -580.564} C_VEL
LIN {X 0,Y 601.345,Z 266.197,A -85,B 0,C 180,E1 -581.771,E2 -581.771} C_VEL
LIN {X 0,Y 601.342,Z 268.487,A -85,B 0,C 180,E1 -582.676,E2 -582.676} C_VEL
LIN {X 0,Y 601.343,Z 270.054,A -85,B 0,C 180,E1 -583.593,E2 -583.593} C_VEL
LIN {X 0,Y 601.334,Z 270.881,A -85,B 0,C 180,E1 -584.526,E2 -584.526} C_VEL
LIN {X 0,Y 601.334,Z 270.907,A -85,B 0,C 180,E1 -585.473,E2 -585.473} C_VEL
LIN {X 0,Y 601.343,Z 270.125,A -85,B 0,C 180,E1 -586.435,E2 -586.435} C_VEL
LIN {X 0,Y 601.342,Z 268.483,A -85,B 0,C 180,E1 -587.416,E2 -587.416} C_VEL
LIN {X 0,Y 601.344,Z 265.894,A -85,B 0,C 180,E1 -588.415,E2 -588.415} C_VEL
LIN {X 0,Y 601.332,Z 262.229,A -85,B 0,C 180,E1 -589.435,E2 -589.435} C_VEL
LIN {X 0,Y 601.385,Z 256.255,A -85,B 0,C 180,E1 -590.674,E2 -590.674} C_VEL
LIN {X 0,Y 601.39,Z 249.662,A -85,B 0,C 180,E1 -591.729,E2 -591.729} C_VEL
LIN {X 0,Y 601.415,Z 241.103,A -85,B 0,C 180,E1 -592.811,E2 -592.811} C_VEL
LIN {X 0,Y 601.44,Z 232.07,A -85,B 0,C 180,E1 -593.734,E2 -593.734} C_VEL
LIN {X 0,Y 601.461,Z 221.561,A -85,B 0,C 180,E1 -594.596,E2 -594.596} C_VEL
LIN {X 0,Y 601.456,Z 211.342,A -85,B 0,C 180,E1 -595.274,E2 -595.274} C_VEL
LIN {X 0,Y 601.46,Z 199.875,A -85,B 0,C 180,E1 -595.883,E2 -595.883} C_VEL
LIN {X 0,Y 601.541,Z 188.668,A -85,B 0,C 180,E1 -596.342,E2 -596.342} C_VEL
LIN {X 0,Y 601.59,Z 176.012,A -85,B 0,C 180,E1 -596.718,E2 -596.718} C_VEL
LIN {X 0,Y 601.424,Z 168.706,A -85,B 0,C 180,E1 -596.876,E2 -596.876} C_VEL
LIN {X 0,Y 601.322,Z 167.669,A -85,B 0,C 180,E1 -596.912,E2 -596.912} C_VEL
LIN {X 0,Y 601.342,Z 163.545,A -85,B 0,C 180,E1 -599.865,E2 -599.865} C_VEL
LIN {X 0,Y 601.329,Z 159.39,A -85,B 0,C 180,E1 -602.883,E2 -602.883} C_VEL
LIN {X 0,Y 601.327,Z 155.366,A -85,B 0,C 180,E1 -605.854,E2 -605.854} C_VEL
LIN {X 0,Y 601.304,Z 151.512,A -85,B 0,C 180,E1 -608.757,E2 -608.757} C_VEL
LIN {X 0,Y 601.306,Z 148.405,A -85,B 0,C 180,E1 -611.211,E2 -611.211} C_VEL
LIN {X 0,Y 601.362,Z 145.333,A -85,B 0,C 180,E1 -613.711,E2 -613.711} C_VEL
LIN {X 0,Y 601.347,Z 141.995,A -85,B 0,C 180,E1 -616.482,E2 -616.482} C_VEL
LIN {X 0,Y 601.386,Z 138.626,A -85,B 0,C 180,E1 -619.223,E2 -619.223} C_VEL
LIN {X 0,Y 601.399,Z 137.804,A -85,B 0,C 180,E1 -619.904,E2 -619.904} C_VEL
LIN {X 0,Y 601.44,Z 137.571,A -85,B 0,C 180,E1 -622.615,E2 -622.615} C_VEL
LIN {X 0,Y 601.419,Z 137.573,A -85,B 0,C 180,E1 -625.308,E2 -625.308} C_VEL
LIN {X 0,Y 601.437,Z 137.568,A -85,B 0,C 180,E1 -627.991,E2 -627.991} C_VEL
LIN {X 0,Y 601.437,Z 137.568,A -85,B 0,C 180,E1 -630.669,E2 -630.669} C_VEL
LIN {X 0,Y 601.422,Z 137.571,A -85,B 0,C 180,E1 -633.349,E2 -633.349} C_VEL
LIN {X 0,Y 601.436,Z 137.572,A -85,B 0,C 180,E1 -636.037,E2 -636.037} C_VEL
LIN {X 0,Y 601.41,Z 137.572,A -85,B 0,C 180,E1 -638.738,E2 -638.738} C_VEL
LIN {X 0,Y 601.433,Z 137.569,A -85,B 0,C 180,E1 -641.458,E2 -641.458} C_VEL
LIN {X 0,Y 601.417,Z 137.572,A -85,B 0,C 180,E1 -644.205,E2 -644.205} C_VEL
LIN {X 0,Y 601.429,Z 137.572,A -85,B 0,C 180,E1 -646.986,E2 -646.986} C_VEL
LIN {X 0,Y 601.406,Z 137.572,A -85,B 0,C 180,E1 -649.809,E2 -649.809} C_VEL
LIN {X 0,Y 601.41,Z 137.573,A -85,B 0,C 180,E1 -652.683,E2 -652.683} C_VEL
LIN {X 0,Y 601.395,Z 137.574,A -85,B 0,C 180,E1 -654.879,E2 -654.879} C_VEL
LIN {X 0,Y 601.414,Z 137.573,A -85,B 0,C 180,E1 -657.868,E2 -657.868} C_VEL
LIN {X 0,Y 601.446,Z 137.571,A -85,B 0,C 180,E1 -660.163,E2 -660.163} C_VEL
LIN {X 0,Y 601.428,Z 137.57,A -85,B 0,C 180,E1 -663.313,E2 -663.313} C_VEL
LIN {X 0,Y 601.395,Z 137.577,A -85,B 0,C 180,E1 -666.26,E2 -666.26} C_VEL
LIN {X 0,Y 601.427,Z 137.572,A -85,B 0,C 180,E1 -668.471,E2 -668.471} C_VEL
LIN {X 0,Y 601.412,Z 137.574,A -85,B 0,C 180,E1 -670.875,E2 -670.875} C_VEL
LIN {X 0,Y 601.427,Z 137.572,A -85,B 0,C 180,E1 -673.586,E2 -673.586} C_VEL
LIN {X 0,Y 601.427,Z 137.569,A -85,B 0,C 180,E1 -676.428,E2 -676.428} C_VEL
LIN {X 0,Y 601.414,Z 137.575,A -85,B 0,C 180,E1 -679.427,E2 -679.427} C_VEL
LIN {X 0,Y 601.425,Z 137.572,A -85,B 0,C 180,E1 -681.733,E2 -681.733} C_VEL
LIN {X 0,Y 601.389,Z 137.578,A -85,B 0,C 180,E1 -684.246,E2 -684.246} C_VEL
LIN {X 0,Y 601.414,Z 137.575,A -85,B 0,C 180,E1 -686.686,E2 -686.686} C_VEL
LIN {X 0,Y 601.423,Z 137.573,A -85,B 0,C 180,E1 -689.059,E2 -689.059} C_VEL
LIN {X 0,Y 601.435,Z 137.571,A -85,B 0,C 180,E1 -691.374,E2 -691.374} C_VEL
LIN {X 0,Y 601.411,Z 137.574,A -85,B 0,C 180,E1 -694.133,E2 -694.133} C_VEL
LIN {X 0,Y 601.415,Z 137.573,A -85,B 0,C 180,E1 -696.59,E2 -696.59} C_VEL
LIN {X 0,Y 601.42,Z 137.57,A -85,B 0,C 180,E1 -699.478,E2 -699.478} C_VEL
LIN {X 0,Y 601.398,Z 137.573,A -85,B 0,C 180,E1 -701.608,E2 -701.608} C_VEL
LIN {X 0,Y 601.42,Z 137.571,A -85,B 0,C 180,E1 -704.409,E2 -704.409} C_VEL
LIN {X 0,Y 601.417,Z 137.574,A -85,B 0,C 180,E1 -707.172,E2 -707.172} C_VEL
LIN {X 0,Y 601.438,Z 137.569,A -85,B 0,C 180,E1 -709.905,E2 -709.905} C_VEL
LIN {X 0,Y 601.408,Z 137.572,A -85,B 0,C 180,E1 -712.615,E2 -712.615} C_VEL
LIN {X 0,Y 601.414,Z 137.571,A -85,B 0,C 180,E1 -715.308,E2 -715.308} C_VEL
LIN {X 0,Y 601.436,Z 137.571,A -85,B 0,C 180,E1 -717.991,E2 -717.991} C_VEL
LIN {X 0,Y 601.449,Z 137.569,A -85,B 0,C 180,E1 -720.67,E2 -720.67} C_VEL
LIN {X 0,Y 601.426,Z 137.57,A -85,B 0,C 180,E1 -723.35,E2 -723.35} C_VEL
LIN {X 0,Y 601.423,Z 137.57,A -85,B 0,C 180,E1 -726.037,E2 -726.037} C_VEL
LIN {X 0,Y 601.409,Z 137.573,A -85,B 0,C 180,E1 -728.738,E2 -728.738} C_VEL
LIN {X 0,Y 601.436,Z 137.571,A -85,B 0,C 180,E1 -731.458,E2 -731.458} C_VEL
LIN {X 0,Y 601.418,Z 137.571,A -85,B 0,C 180,E1 -734.206,E2 -734.206} C_VEL
LIN {X 0,Y 601.413,Z 137.571,A -85,B 0,C 180,E1 -736.987,E2 -736.987} C_VEL
LIN {X 0,Y 601.402,Z 137.576,A -85,B 0,C 180,E1 -739.81,E2 -739.81} C_VEL
LIN {X 0,Y 601.413,Z 137.571,A -85,B 0,C 180,E1 -742.683,E2 -742.683} C_VEL
LIN {X 0,Y 601.401,Z 137.574,A -85,B 0,C 180,E1 -744.879,E2 -744.879} C_VEL
LIN {X 0,Y 601.424,Z 137.571,A -85,B 0,C 180,E1 -747.364,E2 -747.364} C_VEL
LIN {X 0,Y 601.403,Z 137.572,A -85,B 0,C 180,E1 -750.144,E2 -750.144} C_VEL
LIN {X 0,Y 601.412,Z 137.572,A -85,B 0,C 180,E1 -752.714,E2 -752.714} C_VEL
LIN {X 0,Y 601.398,Z 137.573,A -85,B 0,C 180,E1 -755.112,E2 -755.112} C_VEL
LIN {X 0,Y 601.439,Z 137.568,A -85,B 0,C 180,E1 -757.419,E2 -757.419} C_VEL
LIN {X 0,Y 601.402,Z 137.573,A -85,B 0,C 180,E1 -759.996,E2 -759.996} C_VEL
LIN {X 0,Y 601.409,Z 137.574,A -85,B 0,C 180,E1 -762.671,E2 -762.671} C_VEL
LIN {X 0,Y 601.401,Z 137.573,A -85,B 0,C 180,E1 -765.48,E2 -765.48} C_VEL
LIN {X 0,Y 601.421,Z 137.57,A -85,B 0,C 180,E1 -768.408,E2 -768.408} C_VEL
LIN {X 0,Y 601.435,Z 137.57,A -85,B 0,C 180,E1 -770.875,E2 -770.875} C_VEL
LIN {X 0,Y 601.404,Z 137.574,A -85,B 0,C 180,E1 -773.417,E2 -773.417} C_VEL
LIN {X 0,Y 601.421,Z 137.686,A -85,B 0,C 180,E1 -774.158,E2 -774.158} C_VEL
LIN {X 0,Y 601.541,Z 143.795,A -85,B 0,C 180,E1 -776.049,E2 -776.049} C_VEL
LIN {X 0,Y 601.518,Z 153.86,A -85,B 0,C 180,E1 -779.064,E2 -779.064} C_VEL
LIN {X 0,Y 601.47,Z 161.803,A -85,B 0,C 180,E1 -781.375,E2 -781.375} C_VEL
LIN {X 0,Y 601.481,Z 171.451,A -85,B 0,C 180,E1 -784.12,E2 -784.12} C_VEL
LIN {X 0,Y 601.464,Z 180.338,A -85,B 0,C 180,E1 -786.592,E2 -786.592} C_VEL
LIN {X 0,Y 601.431,Z 190.929,A -85,B 0,C 180,E1 -789.478,E2 -789.478} C_VEL
LIN {X 0,Y 601.406,Z 201.521,A -85,B 0,C 180,E1 -792.312,E2 -792.312} C_VEL
LIN {X 0,Y 601.367,Z 212.112,A -85,B 0,C 180,E1 -795.102,E2 -795.102} C_VEL
LIN {X 0,Y 601.343,Z 221.379,A -85,B 0,C 180,E1 -797.513,E2 -797.513} C_VEL
LIN {X 0,Y 601.375,Z 223.53,A -85,B 0,C 180,E1 -798.071,E2 -798.071} C_VEL
LIN {X 0,Y 601.619,Z 235.27,A -85,B 0,C 180,E1 -798.311,E2 -798.311} C_VEL
LIN {X 0,Y 601.534,Z 248.348,A -85,B 0,C 180,E1 -798.691,E2 -798.691} C_VEL
LIN {X 0,Y 601.482,Z 259.243,A -85,B 0,C 180,E1 -799.132,E2 -799.132} C_VEL
LIN {X 0,Y 601.478,Z 270.757,A -85,B 0,C 180,E1 -799.736,E2 -799.736} C_VEL
LIN {X 0,Y 601.462,Z 282.253,A -85,B 0,C 180,E1 -800.5,E2 -800.5} C_VEL
LIN {X 0,Y 601.436,Z 291.537,A -85,B 0,C 180,E1 -801.262,E2 -801.262} C_VEL
LIN {X 0,Y 601.4,Z 299.99,A -85,B 0,C 180,E1 -802.108,E2 -802.108} C_VEL
LIN {X 0,Y 601.382,Z 308.236,A -85,B 0,C 180,E1 -803.12,E2 -803.12} C_VEL
LIN {X 0,Y 601.373,Z 314.877,A -85,B 0,C 180,E1 -804.131,E2 -804.131} C_VEL
LIN {X 0,Y 601.336,Z 320.95,A -85,B 0,C 180,E1 -805.307,E2 -805.307} C_VEL
LIN {X 0,Y 601.368,Z 324.896,A -85,B 0,C 180,E1 -806.315,E2 -806.315} C_VEL
LIN {X 0,Y 601.325,Z 327.809,A -85,B 0,C 180,E1 -807.321,E2 -807.321} C_VEL
LIN {X 0,Y 601.343,Z 329.202,A -85,B 0,C 180,E1 -807.991,E2 -807.991} C_VEL
LIN {X 0,Y 601.339,Z 330.784,A -85,B 0,C 180,E1 -809.33,E2 -809.33} C_VEL
LIN {X 0,Y 601.335,Z 331,A -85,B 0,C 180,E1 -810,E2 -810} C_VEL
LIN {X 0,Y 601.347,Z 330.184,A -85,B 0,C 180,E1 -811.339,E2 -811.339} C_VEL
LIN {X 0,Y 601.343,Z 329.201,A -85,B 0,C 180,E1 -812.009,E2 -812.009} C_VEL
LIN {X 0,Y 601.325,Z 327.809,A -85,B 0,C 180,E1 -812.68,E2 -812.68} C_VEL
LIN {X 0,Y 601.368,Z 324.896,A -85,B 0,C 180,E1 -813.685,E2 -813.685} C_VEL
LIN {X 0,Y 601.336,Z 320.949,A -85,B 0,C 180,E1 -814.693,E2 -814.693} C_VEL
LIN {X 0,Y 601.373,Z 314.876,A -85,B 0,C 180,E1 -815.869,E2 -815.869} C_VEL
LIN {X 0,Y 601.382,Z 308.234,A -85,B 0,C 180,E1 -816.88,E2 -816.88} C_VEL
LIN {X 0,Y 601.4,Z 299.988,A -85,B 0,C 180,E1 -817.892,E2 -817.892} C_VEL
LIN {X 0,Y 601.436,Z 291.535,A -85,B 0,C 180,E1 -818.738,E2 -818.738} C_VEL
LIN {X 0,Y 601.449,Z 281.089,A -85,B 0,C 180,E1 -819.585,E2 -819.585} C_VEL
LIN {X 0,Y 601.478,Z 270.753,A -85,B 0,C 180,E1 -820.264,E2 -820.264} C_VEL
LIN {X 0,Y 601.483,Z 259.233,A -85,B 0,C 180,E1 -820.869,E2 -820.869} C_VEL
LIN {X 0,Y 601.527,Z 246.332,A -85,B 0,C 180,E1 -821.375,E2 -821.375} C_VEL
LIN {X 0,Y 601.617,Z 233.431,A -85,B 0,C 180,E1 -821.732,E2 -821.732} C_VEL
LIN {X 0,Y 601.376,Z 223.53,A -85,B 0,C 180,E1 -821.93,E2 -821.93} C_VEL
LIN {X 0,Y 601.372,Z 213.435,A -85,B 0,C 180,E1 -824.552,E2 -824.552} C_VEL
LIN {X 0,Y 601.397,Z 202.844,A -85,B 0,C 180,E1 -827.337,E2 -827.337} C_VEL
LIN {X 0,Y 601.424,Z 192.252,A -85,B 0,C 180,E1 -830.165,E2 -830.165} C_VEL
LIN {X 0,Y 601.433,Z 182.985,A -85,B 0,C 180,E1 -832.682,E2 -832.682} C_VEL
LIN {X 0,Y 601.459,Z 173.718,A -85,B 0,C 180,E1 -835.246,E2 -835.246} C_VEL
LIN {X 0,Y 601.503,Z 164.45,A -85,B 0,C 180,E1 -837.863,E2 -837.863} C_VEL
LIN {X 0,Y 601.483,Z 155.183,A -85,B 0,C 180,E1 -840.549,E2 -840.549} C_VEL
LIN {X 0,Y 601.516,Z 147.837,A -85,B 0,C 180,E1 -842.729,E2 -842.729} C_VEL
LIN {X 0,Y 601.582,Z 139.922,A -85,B 0,C 180,E1 -845.137,E2 -845.137} C_VEL
LIN {X 0,Y 601.423,Z 137.573,A -85,B 0,C 180,E1 -845.932,E2 -845.932} C_VEL
LIN {X 0,Y 601.437,Z 137.57,A -85,B 0,C 180,E1 -848.471,E2 -848.471} C_VEL
LIN {X 0,Y 601.427,Z 137.571,A -85,B 0,C 180,E1 -851.593,E2 -851.593} C_VEL
LIN {X 0,Y 601.43,Z 137.571,A -85,B 0,C 180,E1 -854.535,E2 -854.535} C_VEL
LIN {X 0,Y 601.412,Z 137.574,A -85,B 0,C 180,E1 -857.41,E2 -857.41} C_VEL
LIN {X 0,Y 601.447,Z 137.57,A -85,B 0,C 180,E1 -860.464,E2 -860.464} C_VEL
LIN {X 0,Y 601.408,Z 137.575,A -85,B 0,C 180,E1 -863.417,E2 -863.417} C_VEL
LIN {X 0,Y 601.437,Z 137.57,A -85,B 0,C 180,E1 -866.064,E2 -866.064} C_VEL
LIN {X 0,Y 601.435,Z 137.571,A -85,B 0,C 180,E1 -868.544,E2 -868.544} C_VEL
LIN {X 0,Y 601.435,Z 137.572,A -85,B 0,C 180,E1 -871.373,E2 -871.373} C_VEL
LIN {X 0,Y 601.403,Z 137.575,A -85,B 0,C 180,E1 -873.636,E2 -873.636} C_VEL
LIN {X 0,Y 601.419,Z 137.573,A -85,B 0,C 180,E1 -876.589,E2 -876.589} C_VEL
LIN {X 0,Y 601.432,Z 137.573,A -85,B 0,C 180,E1 -879.478,E2 -879.478} C_VEL
LIN {X 0,Y 601.396,Z 137.575,A -85,B 0,C 180,E1 -882.311,E2 -882.311} C_VEL
LIN {X 0,Y 601.414,Z 137.574,A -85,B 0,C 180,E1 -884.408,E2 -884.408} C_VEL
LIN {X 0,Y 601.42,Z 137.572,A -85,B 0,C 180,E1 -887.172,E2 -887.172} C_VEL
LIN {X 0,Y 601.441,Z 137.569,A -85,B 0,C 180,E1 -889.905,E2 -889.905} C_VEL
LIN {X 0,Y 601.443,Z 137.571,A -85,B 0,C 180,E1 -892.615,E2 -892.615} C_VEL
LIN {X 0,Y 601.422,Z 137.572,A -85,B 0,C 180,E1 -895.308,E2 -895.308} C_VEL
LIN {X 0,Y 601.438,Z 137.57,A -85,B 0,C 180,E1 -897.991,E2 -897.991} C_VEL
LIN {X 0,Y 601.456,Z 137.57,A -85,B 0,C 180,E1 -900.669,E2 -900.669} C_VEL
LIN {X 0,Y 601.423,Z 137.571,A -85,B 0,C 180,E1 -903.349,E2 -903.349} C_VEL
LIN {X 0,Y 601.421,Z 137.572,A -85,B 0,C 180,E1 -906.037,E2 -906.037} C_VEL
LIN {X 0,Y 601.411,Z 137.575,A -85,B 0,C 180,E1 -908.738,E2 -908.738} C_VEL
LIN {X 0,Y 601.399,Z 137.807,A -85,B 0,C 180,E1 -910.095,E2 -910.095} C_VEL
LIN {X 0,Y 601.353,Z 140.628,A -85,B 0,C 180,E1 -912.349,E2 -912.349} C_VEL
LIN {X 0,Y 600.689,Z 141.371,A -85,B 0,C 180,E1 -912.904,E2 -912.904} C_VEL
LIN {X 0,Y 597.831,Z 142.717,A -85,B 0,C 180,E1 -913.803,E2 -913.803} C_VEL
LIN {X 0,Y 595.411,Z 143.801,A -85,B 0,C 180,E1 -914.526,E2 -914.526} C_VEL
LIN {X 0,Y 594.367,Z 144.56,A -85,B 0,C 180,E1 -915.085,E2 -915.085} C_VEL
LIN {X 0,Y 594.28,Z 144.794,A -85,B 0,C 180,E1 -915.274,E2 -915.274} C_VEL
LIN {X 0,Y 594.281,Z 147.927,A -85,B 0,C 180,E1 -917.907,E2 -917.907} C_VEL
LIN {X 0,Y 594.265,Z 151.213,A -85,B 0,C 180,E1 -920.78,E2 -920.78} C_VEL
LIN {X 0,Y 594.223,Z 155.016,A -85,B 0,C 180,E1 -923.711,E2 -923.711} C_VEL
LIN {X 0,Y 594.227,Z 158.05,A -85,B 0,C 180,E1 -925.991,E2 -925.991} C_VEL
LIN {X 0,Y 594.222,Z 161.078,A -85,B 0,C 180,E1 -928.235,E2 -928.235} C_VEL
LIN {X 0,Y 594.23,Z 164.264,A -85,B 0,C 180,E1 -930.568,E2 -930.568} C_VEL
LIN {X 0,Y 594.25,Z 167.685,A -85,B 0,C 180,E1 -933.046,E2 -933.046} C_VEL
LIN {X 0,Y 594.668,Z 172.804,A -85,B 0,C 180,E1 -933.159,E2 -933.159} C_VEL
LIN {X 0,Y 594.594,Z 185.062,A -85,B 0,C 180,E1 -933.493,E2 -933.493} C_VEL
LIN {X 0,Y 594.499,Z 197.477,A -85,B 0,C 180,E1 -933.969,E2 -933.969} C_VEL
LIN {X 0,Y 594.467,Z 209.352,A -85,B 0,C 180,E1 -934.574,E2 -934.574} C_VEL
LIN {X 0,Y 594.46,Z 220.981,A -85,B 0,C 180,E1 -935.338,E2 -935.338} C_VEL
LIN {X 0,Y 594.409,Z 230.767,A -85,B 0,C 180,E1 -936.135,E2 -936.135} C_VEL
LIN {X 0,Y 594.348,Z 238.758,A -85,B 0,C 180,E1 -936.924,E2 -936.924} C_VEL
LIN {X 0,Y 594.298,Z 247.251,A -85,B 0,C 180,E1 -937.947,E2 -937.947} C_VEL
LIN {X 0,Y 594.273,Z 254.435,A -85,B 0,C 180,E1 -939.031,E2 -939.031} C_VEL
LIN {X 0,Y 594.284,Z 260.247,A -85,B 0,C 180,E1 -940.142,E2 -940.142} C_VEL
LIN {X 0,Y 594.234,Z 264.192,A -85,B 0,C 180,E1 -941.117,E2 -941.117} C_VEL
LIN {X 0,Y 594.27,Z 267.926,A -85,B 0,C 180,E1 -942.384,E2 -942.384} C_VEL
LIN {X 0,Y 594.245,Z 269.686,A -85,B 0,C 180,E1 -943.31,E2 -943.31} C_VEL
LIN {X 0,Y 594.23,Z 270.704,A -85,B 0,C 180,E1 -944.25,E2 -944.25} C_VEL
LIN {X 0,Y 594.22,Z 270.97,A -85,B 0,C 180,E1 -945.205,E2 -945.205} C_VEL
LIN {X 0,Y 594.235,Z 270.446,A -85,B 0,C 180,E1 -946.173,E2 -946.173} C_VEL
LIN {X 0,Y 594.247,Z 269.066,A -85,B 0,C 180,E1 -947.16,E2 -947.16} C_VEL
LIN {X 0,Y 594.24,Z 265.68,A -85,B 0,C 180,E1 -948.524,E2 -948.524} C_VEL
LIN {X 0,Y 594.252,Z 262.5,A -85,B 0,C 180,E1 -949.423,E2 -949.423} C_VEL
LIN {X 0,Y 594.293,Z 257.367,A -85,B 0,C 180,E1 -950.532,E2 -950.532} C_VEL
LIN {X 0,Y 594.297,Z 250.535,A -85,B 0,C 180,E1 -951.679,E2 -951.679} C_VEL
LIN {X 0,Y 594.333,Z 243.228,A -85,B 0,C 180,E1 -952.658,E2 -952.658} C_VEL
LIN {X 0,Y 594.412,Z 234.12,A -85,B 0,C 180,E1 -953.64,E2 -953.64} C_VEL
LIN {X 0,Y 594.419,Z 224.419,A -85,B 0,C 180,E1 -954.491,E2 -954.491} C_VEL
LIN {X 0,Y 594.442,Z 214.252,A -85,B 0,C 180,E1 -955.218,E2 -955.218} C_VEL
LIN {X 0,Y 594.458,Z 203.183,A -85,B 0,C 180,E1 -955.85,E2 -955.85} C_VEL
LIN {X 0,Y 594.559,Z 190.606,A -85,B 0,C 180,E1 -956.403,E2 -956.403} C_VEL
LIN {X 0,Y 594.643,Z 177.752,A -85,B 0,C 180,E1 -956.814,E2 -956.814} C_VEL
LIN {X 0,Y 594.473,Z 169.319,A -85,B 0,C 180,E1 -957.005,E2 -957.005} C_VEL
LIN {X 0,Y 594.236,Z 167.666,A -85,B 0,C 180,E1 -957.058,E2 -957.058} C_VEL
LIN {X 0,Y 594.236,Z 164.026,A -85,B 0,C 180,E1 -959.696,E2 -959.696} C_VEL
LIN {X 0,Y 594.259,Z 160.159,A -85,B 0,C 180,E1 -962.533,E2 -962.533} C_VEL
LIN {X 0,Y 594.237,Z 156.051,A -85,B 0,C 180,E1 -965.598,E2 -965.598} C_VEL
LIN {X 0,Y 594.212,Z 152.248,A -85,B 0,C 180,E1 -968.491,E2 -968.491} C_VEL
LIN {X 0,Y 594.254,Z 149.145,A -85,B 0,C 180,E1 -971.106,E2 -971.106} C_VEL
LIN {X 0,Y 594.308,Z 146.158,A -85,B 0,C 180,E1 -973.512,E2 -973.512} C_VEL
LIN {X 0,Y 594.272,Z 142.758,A -85,B 0,C 180,E1 -976.318,E2 -976.318} C_VEL
LIN {X 0,Y 594.311,Z 139.389,A -85,B 0,C 180,E1 -979.093,E2 -979.093} C_VEL
LIN {X 0,Y 594.344,Z 138.571,A -85,B 0,C 180,E1 -979.783,E2 -979.783} C_VEL
LIN {X 0,Y 594.393,Z 138.448,A -85,B 0,C 180,E1 -982.527,E2 -982.527} C_VEL
LIN {X 0,Y 594.388,Z 138.449,A -85,B 0,C 180,E1 -985.252,E2 -985.252} C_VEL
LIN {X 0,Y 594.406,Z 138.444,A -85,B 0,C 180,E1 -987.967,E2 -987.967} C_VEL
LIN {X 0,Y 594.41,Z 138.444,A -85,B 0,C 180,E1 -990.677,E2 -990.677} C_VEL
LIN {X 0,Y 594.374,Z 138.45,A -85,B 0,C 180,E1 -993.389,E2 -993.389} C_VEL
LIN {X 0,Y 594.382,Z 138.45,A -85,B 0,C 180,E1 -996.109,E2 -996.109} C_VEL
LIN {X 0,Y 594.377,Z 138.448,A -85,B 0,C 180,E1 -998.842,E2 -998.842} C_VEL
LIN {X 0,Y 594.392,Z 138.446,A -85,B 0,C 180,E1 -1001.596,E2 -1001.596} C_VEL
LIN {X 0,Y 594.387,Z 138.45,A -85,B 0,C 180,E1 -1004.377,E2 -1004.377} C_VEL
LIN {X 0,Y 594.388,Z 138.447,A -85,B 0,C 180,E1 -1007.193,E2 -1007.193} C_VEL
LIN {X 0,Y 594.376,Z 138.448,A -85,B 0,C 180,E1 -1010.054,E2 -1010.054} C_VEL
LIN {X 0,Y 594.364,Z 138.453,A -85,B 0,C 180,E1 -1012.967,E2 -1012.967} C_VEL
LIN {X 0,Y 594.369,Z 138.451,A -85,B 0,C 180,E1 -1015.193,E2 -1015.193} C_VEL
LIN {X 0,Y 594.383,Z 138.449,A -85,B 0,C 180,E1 -1017.527,E2 -1017.527} C_VEL
LIN {X 0,Y 594.397,Z 138.447,A -85,B 0,C 180,E1 -1020.331,E2 -1020.331} C_VEL
LIN {X 0,Y 594.377,Z 138.448,A -85,B 0,C 180,E1 -1022.95,E2 -1022.95} C_VEL
LIN {X 0,Y 594.348,Z 138.452,A -85,B 0,C 180,E1 -1025.409,E2 -1025.409} C_VEL
LIN {X 0,Y 594.379,Z 138.447,A -85,B 0,C 180,E1 -1027.941,E2 -1027.941} C_VEL
LIN {X 0,Y 594.374,Z 138.45,A -85,B 0,C 180,E1 -1030.822,E2 -1030.822} C_VEL
LIN {X 0,Y 594.366,Z 138.452,A -85,B 0,C 180,E1 -1033.3,E2 -1033.3} C_VEL
LIN {X 0,Y 594.366,Z 138.45,A -85,B 0,C 180,E1 -1036.161,E2 -1036.161} C_VEL
LIN {X 0,Y 594.379,Z 138.449,A -85,B 0,C 180,E1 -1039.178,E2 -1039.178} C_VEL
LIN {X 0,Y 594.389,Z 138.448,A -85,B 0,C 180,E1 -1042.06,E2 -1042.06} C_VEL
LIN {X 0,Y 594.361,Z 138.45,A -85,B 0,C 180,E1 -1044.675,E2 -1044.675} C_VEL
LIN {X 0,Y 594.375,Z 138.448,A -85,B 0,C 180,E1 -1047.089,E2 -1047.089} C_VEL
LIN {X 0,Y 594.37,Z 138.448,A -85,B 0,C 180,E1 -1049.675,E2 -1049.675} C_VEL
LIN {X 0,Y 594.375,Z 138.45,A -85,B 0,C 180,E1 -1052.54,E2 -1052.54} C_VEL
LIN {X 0,Y 594.377,Z 138.448,A -85,B 0,C 180,E1 -1054.807,E2 -1054.807} C_VEL
LIN {X 0,Y 594.364,Z 138.45,A -85,B 0,C 180,E1 -1057.265,E2 -1057.265} C_VEL
LIN {X 0,Y 594.371,Z 138.452,A -85,B 0,C 180,E1 -1059.947,E2 -1059.947} C_VEL
LIN {X 0,Y 594.375,Z 138.448,A -85,B 0,C 180,E1 -1062.807,E2 -1062.807} C_VEL
LIN {X 0,Y 594.389,Z 138.448,A -85,B 0,C 180,E1 -1065.827,E2 -1065.827} C_VEL
LIN {X 0,Y 594.381,Z 138.451,A -85,B 0,C 180,E1 -1068.404,E2 -1068.404} C_VEL
LIN {X 0,Y 594.377,Z 138.448,A -85,B 0,C 180,E1 -1071.158,E2 -1071.158} C_VEL
LIN {X 0,Y 594.376,Z 138.448,A -85,B 0,C 180,E1 -1073.892,E2 -1073.892} C_VEL
LIN {X 0,Y 594.386,Z 138.448,A -85,B 0,C 180,E1 -1076.611,E2 -1076.611} C_VEL
LIN {X 0,Y 594.426,Z 138.445,A -85,B 0,C 180,E1 -1079.323,E2 -1079.323} C_VEL
LIN {X 0,Y 594.406,Z 138.445,A -85,B 0,C 180,E1 -1082.033,E2 -1082.033} C_VEL
LIN {X 0,Y 594.382,Z 138.447,A -85,B 0,C 180,E1 -1084.748,E2 -1084.748} C_VEL
LIN {X 0,Y 594.371,Z 138.449,A -85,B 0,C 180,E1 -1087.474,E2 -1087.474} C_VEL
LIN {X 0,Y 594.393,Z 138.449,A -85,B 0,C 180,E1 -1090.216,E2 -1090.216} C_VEL
LIN {X 0,Y 594.366,Z 138.449,A -85,B 0,C 180,E1 -1092.983,E2 -1092.983} C_VEL
LIN {X 0,Y 594.37,Z 138.449,A -85,B 0,C 180,E1 -1095.781,E2 -1095.781} C_VEL
LIN {X 0,Y 594.387,Z 138.45,A -85,B 0,C 180,E1 -1098.618,E2 -1098.618} C_VEL
LIN {X 0,Y 594.369,Z 138.449,A -85,B 0,C 180,E1 -1101.504,E2 -1101.504} C_VEL
LIN {X 0,Y 594.391,Z 138.448,A -85,B 0,C 180,E1 -1104.446,E2 -1104.446} C_VEL
LIN {X 0,Y 594.387,Z 138.447,A -85,B 0,C 180,E1 -1106.7,E2 -1106.7} C_VEL
LIN {X 0,Y 594.383,Z 138.447,A -85,B 0,C 180,E1 -1108.999,E2 -1108.999} C_VEL
LIN {X 0,Y 594.393,Z 138.447,A -85,B 0,C 180,E1 -1111.645,E2 -1111.645} C_VEL
LIN {X 0,Y 594.378,Z 138.449,A -85,B 0,C 180,E1 -1114.58,E2 -1114.58} C_VEL
LIN {X 0,Y 594.392,Z 138.447,A -85,B 0,C 180,E1 -1117.609,E2 -1117.609} C_VEL
LIN {X 0,Y 594.37,Z 138.45,A -85,B 0,C 180,E1 -1120.567,E2 -1120.567} C_VEL
LIN {X 0,Y 594.368,Z 138.448,A -85,B 0,C 180,E1 -1123.3,E2 -1123.3} C_VEL
LIN {X 0,Y 594.362,Z 138.451,A -85,B 0,C 180,E1 -1126.162,E2 -1126.162} C_VEL
LIN {X 0,Y 594.379,Z 138.448,A -85,B 0,C 180,E1 -1128.536,E2 -1128.536} C_VEL
LIN {X 0,Y 594.38,Z 138.451,A -85,B 0,C 180,E1 -1131.297,E2 -1131.297} C_VEL
LIN {X 0,Y 594.393,Z 138.635,A -85,B 0,C 180,E1 -1133.968,E2 -1133.968} C_VEL
LIN {X 0,Y 594.604,Z 143.269,A -85,B 0,C 180,E1 -1135.435,E2 -1135.435} C_VEL
LIN {X 0,Y 594.545,Z 149.888,A -85,B 0,C 180,E1 -1137.463,E2 -1137.463} C_VEL
LIN {X 0,Y 594.515,Z 157.193,A -85,B 0,C 180,E1 -1139.651,E2 -1139.651} C_VEL
LIN {X 0,Y 594.511,Z 167.099,A -85,B 0,C 180,E1 -1142.546,E2 -1142.546} C_VEL
LIN {X 0,Y 594.464,Z 176.366,A -85,B 0,C 180,E1 -1145.185,E2 -1145.185} C_VEL
LIN {X 0,Y 594.411,Z 186.958,A -85,B 0,C 180,E1 -1148.134,E2 -1148.134} C_VEL
LIN {X 0,Y 594.363,Z 197.746,A -85,B 0,C 180,E1 -1151.077,E2 -1151.077} C_VEL
LIN {X 0,Y 594.312,Z 208.14,A -85,B 0,C 180,E1 -1153.865,E2 -1153.865} C_VEL
LIN {X 0,Y 594.332,Z 218.731,A -85,B 0,C 180,E1 -1156.668,E2 -1156.668} C_VEL
LIN {X 0,Y 594.286,Z 223.53,A -85,B 0,C 180,E1 -1157.926,E2 -1157.926} C_VEL
LIN {X 0,Y 594.67,Z 229.234,A -85,B 0,C 180,E1 -1158.042,E2 -1158.042} C_VEL
LIN {X 0,Y 594.614,Z 242.498,A -85,B 0,C 180,E1 -1158.366,E2 -1158.366} C_VEL
LIN {X 0,Y 594.531,Z 254.644,A -85,B 0,C 180,E1 -1158.801,E2 -1158.801} C_VEL
LIN {X 0,Y 594.475,Z 266.209,A -85,B 0,C 180,E1 -1159.355,E2 -1159.355} C_VEL
LIN {X 0,Y 594.465,Z 277.477,A -85,B 0,C 180,E1 -1160.043,E2 -1160.043} C_VEL
LIN {X 0,Y 594.406,Z 287.648,A -85,B 0,C 180,E1 -1160.815,E2 -1160.815} C_VEL
LIN {X 0,Y 594.372,Z 296.788,A -85,B 0,C 180,E1 -1161.672,E2 -1161.672} C_VEL
LIN {X 0,Y 594.316,Z 305.691,A -85,B 0,C 180,E1 -1162.697,E2 -1162.697} C_VEL
LIN {X 0,Y 594.281,Z 312.17,A -85,B 0,C 180,E1 -1163.615,E2 -1163.615} C_VEL
LIN {X 0,Y 594.289,Z 317.681,A -85,B 0,C 180,E1 -1164.571,E2 -1164.571} C_VEL
LIN {X 0,Y 594.27,Z 322.371,A -85,B 0,C 180,E1 -1165.591,E2 -1165.591} C_VEL
LIN {X 0,Y 594.267,Z 325.956,A -85,B 0,C 180,E1 -1166.61,E2 -1166.61} C_VEL
LIN {X 0,Y 594.226,Z 327.809,A -85,B 0,C 180,E1 -1167.289,E2 -1167.289} C_VEL
LIN {X 0,Y 594.242,Z 329.202,A -85,B 0,C 180,E1 -1167.967,E2 -1167.967} C_VEL
LIN {X 0,Y 594.239,Z 330.784,A -85,B 0,C 180,E1 -1169.322,E2 -1169.322} C_VEL
LIN {X 0,Y 594.236,Z 331,A -85,B 0,C 180,E1 -1170,E2 -1170} C_VEL
LIN {X 0,Y 594.247,Z 330.184,A -85,B 0,C 180,E1 -1171.355,E2 -1171.355} C_VEL
LIN {X 0,Y 594.242,Z 329.202,A -85,B 0,C 180,E1 -1172.033,E2 -1172.033} C_VEL
LIN {X 0,Y 594.226,Z 327.809,A -85,B 0,C 180,E1 -1172.712,E2 -1172.712} C_VEL
LIN {X 0,Y 594.289,Z 324.896,A -85,B 0,C 180,E1 -1173.729,E2 -1173.729} C_VEL
LIN {X 0,Y 594.241,Z 320.949,A -85,B 0,C 180,E1 -1174.749,E2 -1174.749} C_VEL
LIN {X 0,Y 594.305,Z 314.876,A -85,B 0,C 180,E1 -1175.939,E2 -1175.939} C_VEL
LIN {X 0,Y 594.308,Z 308.234,A -85,B 0,C 180,E1 -1176.962,E2 -1176.962} C_VEL
LIN {X 0,Y 594.359,Z 299.988,A -85,B 0,C 180,E1 -1177.987,E2 -1177.987} C_VEL
LIN {X 0,Y 594.382,Z 291.535,A -85,B 0,C 180,E1 -1178.842,E2 -1178.842} C_VEL
LIN {X 0,Y 594.431,Z 281.09,A -85,B 0,C 180,E1 -1179.7,E2 -1179.7} C_VEL
LIN {X 0,Y 594.454,Z 270.754,A -85,B 0,C 180,E1 -1180.387,E2 -1180.387} C_VEL
LIN {X 0,Y 594.501,Z 258.77,A -85,B 0,C 180,E1 -1181.019,E2 -1181.019} C_VEL
LIN {X 0,Y 594.56,Z 246.487,A -85,B 0,C 180,E1 -1181.505,E2 -1181.505} C_VEL
LIN {X 0,Y 594.676,Z 233.431,A -85,B 0,C 180,E1 -1181.871,E2 -1181.871} C_VEL
LIN {X 0,Y 594.457,Z 224.85,A -85,B 0,C 180,E1 -1182.038,E2 -1182.038} C_VEL
LIN {X 0,Y 594.288,Z 223.53,A -85,B 0,C 180,E1 -1182.074,E2 -1182.074} C_VEL
LIN {X 0,Y 594.306,Z 213.435,A -85,B 0,C 180,E1 -1184.729,E2 -1184.729} C_VEL
LIN {X 0,Y 594.339,Z 202.844,A -85,B 0,C 180,E1 -1187.55,E2 -1187.55} C_VEL
LIN {X 0,Y 594.384,Z 192.252,A -85,B 0,C 180,E1 -1190.415,E2 -1190.415} C_VEL
LIN {X 0,Y 594.438,Z 181.661,A -85,B 0,C 180,E1 -1193.333,E2 -1193.333} C_VEL
LIN {X 0,Y 594.489,Z 172.031,A -85,B 0,C 180,E1 -1196.042,E2 -1196.042} C_VEL
LIN {X 0,Y 594.479,Z 163.148,A -85,B 0,C 180,E1 -1198.601,E2 -1198.601} C_VEL
LIN {X 0,Y 594.585,Z 153.859,A -85,B 0,C 180,E1 -1201.338,E2 -1201.338} C_VEL
LIN {X 0,Y 594.611,Z 145.916,A -85,B 0,C 180,E1 -1203.747,E2 -1203.747} C_VEL
LIN {X 0,Y 594.513,Z 139.296,A -85,B 0,C 180,E1 -1205.815,E2 -1205.815} C_VEL
LIN {X 0,Y 594.372,Z 138.452,A -85,B 0,C 180,E1 -1206.138,E2 -1206.138} C_VEL
LIN {X 0,Y 594.383,Z 138.448,A -85,B 0,C 180,E1 -1208.805,E2 -1208.805} C_VEL
LIN {X 0,Y 594.386,Z 138.448,A -85,B 0,C 180,E1 -1211.848,E2 -1211.848} C_VEL
LIN {X 0,Y 594.369,Z 138.45,A -85,B 0,C 180,E1 -1214.809,E2 -1214.809} C_VEL
LIN {X 0,Y 594.37,Z 138.45,A -85,B 0,C 180,E1 -1217.624,E2 -1217.624} C_VEL
LIN {X 0,Y 594.398,Z 138.449,A -85,B 0,C 180,E1 -1220.321,E2 -1220.321} C_VEL
LIN {X 0,Y 594.388,Z 138.448,A -85,B 0,C 180,E1 -1222.913,E2 -1222.913} C_VEL
LIN {X 0,Y 594.387,Z 138.447,A -85,B 0,C 180,E1 -1225.861,E2 -1225.861} C_VEL
LIN {X 0,Y 594.384,Z 138.448,A -85,B 0,C 180,E1 -1228.65,E2 -1228.65} C_VEL
LIN {X 0,Y 594.388,Z 138.448,A -85,B 0,C 180,E1 -1231.042,E2 -1231.042} C_VEL
LIN {X 0,Y 594.389,Z 138.447,A -85,B 0,C 180,E1 -1233.977,E2 -1233.977} C_VEL
LIN {X 0,Y 594.388,Z 138.449,A -85,B 0,C 180,E1 -1236.296,E2 -1236.296} C_VEL
LIN {X 0,Y 594.407,Z 138.446,A -85,B 0,C 180,E1 -1239.224,E2 -1239.224} C_VEL
LIN {X 0,Y 594.354,Z 138.451,A -85,B 0,C 180,E1 -1242.095,E2 -1242.095} C_VEL
LIN {X 0,Y 594.368,Z 138.45,A -85,B 0,C 180,E1 -1244.219,E2 -1244.219} C_VEL
LIN {X 0,Y 594.385,Z 138.449,A -85,B 0,C 180,E1 -1246.321,E2 -1246.321} C_VEL
LIN {X 0,Y 594.378,Z 138.449,A -85,B 0,C 180,E1 -1249.094,E2 -1249.094} C_VEL
LIN {X 0,Y 594.418,Z 138.444,A -85,B 0,C 180,E1 -1251.843,E2 -1251.843} C_VEL
LIN {X 0,Y 594.398,Z 138.449,A -85,B 0,C 180,E1 -1254.572,E2 -1254.572} C_VEL
LIN {X 0,Y 594.407,Z 138.445,A -85,B 0,C 180,E1 -1257.289,E2 -1257.289} C_VEL
LIN {X 0,Y 594.42,Z 138.444,A -85,B 0,C 180,E1 -1260,E2 -1260} C_VEL
LIN {X 0,Y 594.411,Z 138.447,A -85,B 0,C 180,E1 -1262.71,E2 -1262.71} C_VEL
LIN {X 0,Y 594.389,Z 138.448,A -85,B 0,C 180,E1 -1265.427,E2 -1265.427} C_VEL
LIN {X 0,Y 594.416,Z 138.444,A -85,B 0,C 180,E1 -1268.156,E2 -1268.156} C_VEL
LIN {X 0,Y 594.345,Z 138.629,A -85,B 0,C 180,E1 -1270.216,E2 -1270.216} C_VEL
LIN {X 0,Y 594.294,Z 142.047,A -85,B 0,C 180,E1 -1272.984,E2 -1272.984} C_VEL
LIN {X 0,Y 594.28,Z 144.794,A -85,B 0,C 180,E1 -1275.274,E2 -1275.274} C_VEL
LIN {X 0,Y 593.605,Z 145.527,A -85,B 0,C 180,E1 -1275.836,E2 -1275.836} C_VEL
LIN {X 0,Y 590.739,Z 146.859,A -85,B 0,C 180,E1 -1276.745,E2 -1276.745} C_VEL
LIN {X 0,Y 588.316,Z 147.939,A -85,B 0,C 180,E1 -1277.476,E2 -1277.476} C_VEL
LIN {X 0,Y 587.27,Z 148.702,A -85,B 0,C 180,E1 -1278.041,E2 -1278.041} C_VEL
LIN {X 0,Y 587.181,Z 148.939,A -85,B 0,C 180,E1 -1278.232,E2 -1278.232} C_VEL
LIN {X 0,Y 587.165,Z 152.222,A -85,B 0,C 180,E1 -1281.043,E2 -1281.043} C_VEL
LIN {X 0,Y 587.112,Z 154.792,A -85,B 0,C 180,E1 -1283.267,E2 -1283.267} C_VEL
LIN {X 0,Y 587.136,Z 157.752,A -85,B 0,C 180,E1 -1285.525,E2 -1285.525} C_VEL
LIN {X 0,Y 587.152,Z 160.812,A -85,B 0,C 180,E1 -1287.827,E2 -1287.827} C_VEL
LIN {X 0,Y 587.155,Z 164.386,A -85,B 0,C 180,E1 -1290.479,E2 -1290.479} C_VEL
LIN {X 0,Y 587.148,Z 167.681,A -85,B 0,C 180,E1 -1292.896,E2 -1292.896} C_VEL
LIN {X 0,Y 587.73,Z 173.634,A -85,B 0,C 180,E1 -1293.036,E2 -1293.036} C_VEL
LIN {X 0,Y 587.63,Z 187.272,A -85,B 0,C 180,E1 -1293.429,E2 -1293.429} C_VEL
LIN {X 0,Y 587.541,Z 198.85,A -85,B 0,C 180,E1 -1293.897,E2 -1293.897} C_VEL
LIN {X 0,Y 587.463,Z 209.654,A -85,B 0,C 180,E1 -1294.466,E2 -1294.466} C_VEL
LIN {X 0,Y 587.439,Z 221.044,A -85,B 0,C 180,E1 -1295.225,E2 -1295.225} C_VEL
LIN {X 0,Y 587.354,Z 231.654,A -85,B 0,C 180,E1 -1296.107,E2 -1296.107} C_VEL
LIN {X 0,Y 587.296,Z 240.012,A -85,B 0,C 180,E1 -1296.964,E2 -1296.964} C_VEL
LIN {X 0,Y 587.22,Z 247.893,A -85,B 0,C 180,E1 -1297.951,E2 -1297.951} C_VEL
LIN {X 0,Y 587.208,Z 255.398,A -85,B 0,C 180,E1 -1299.123,E2 -1299.123} C_VEL
LIN {X 0,Y 587.2,Z 261.049,A -85,B 0,C 180,E1 -1300.263,E2 -1300.263} C_VEL
LIN {X 0,Y 587.141,Z 264.564,A -85,B 0,C 180,E1 -1301.173,E2 -1301.173} C_VEL
LIN {X 0,Y 587.19,Z 267.273,A -85,B 0,C 180,E1 -1302.092,E2 -1302.092} C_VEL
LIN {X 0,Y 587.147,Z 269.384,A -85,B 0,C 180,E1 -1303.1,E2 -1303.1} C_VEL
LIN {X 0,Y 587.155,Z 270.604,A -85,B 0,C 180,E1 -1304.096,E2 -1304.096} C_VEL
LIN {X 0,Y 587.143,Z 270.999,A -85,B 0,C 180,E1 -1305.071,E2 -1305.071} C_VEL
LIN {X 0,Y 587.135,Z 270.578,A -85,B 0,C 180,E1 -1306.031,E2 -1306.031} C_VEL
LIN {X 0,Y 587.163,Z 269.4,A -85,B 0,C 180,E1 -1306.979,E2 -1306.979} C_VEL
LIN {X 0,Y 587.165,Z 266.28,A -85,B 0,C 180,E1 -1308.371,E2 -1308.371} C_VEL
LIN {X 0,Y 587.161,Z 263.034,A -85,B 0,C 180,E1 -1309.342,E2 -1309.342} C_VEL
LIN {X 0,Y 587.208,Z 258.815,A -85,B 0,C 180,E1 -1310.313,E2 -1310.313} C_VEL
LIN {X 0,Y 587.232,Z 253.483,A -85,B 0,C 180,E1 -1311.294,E2 -1311.294} C_VEL
LIN {X 0,Y 587.241,Z 246.102,A -85,B 0,C 180,E1 -1312.384,E2 -1312.384} C_VEL
LIN {X 0,Y 587.277,Z 238.416,A -85,B 0,C 180,E1 -1313.301,E2 -1313.301} C_VEL
LIN {X 0,Y 587.374,Z 229.157,A -85,B 0,C 180,E1 -1314.207,E2 -1314.207} C_VEL
LIN {X 0,Y 587.428,Z 218.605,A -85,B 0,C 180,E1 -1315.045,E2 -1315.045} C_VEL
LIN {X 0,Y 587.473,Z 206.773,A -85,B 0,C 180,E1 -1315.787,E2 -1315.787} C_VEL
LIN {X 0,Y 587.545,Z 195.077,A -85,B 0,C 180,E1 -1316.36,E2 -1316.36} C_VEL
LIN {X 0,Y 587.672,Z 182.245,A -85,B 0,C 180,E1 -1316.826,E2 -1316.826} C_VEL
LIN {X 0,Y 587.512,Z 170.309,A -85,B 0,C 180,E1 -1317.13,E2 -1317.13} C_VEL
LIN {X 0,Y 587.145,Z 167.672,A -85,B 0,C 180,E1 -1317.201,E2 -1317.201} C_VEL
LIN {X 0,Y 587.153,Z 164.103,A -85,B 0,C 180,E1 -1319.819,E2 -1319.819} C_VEL
LIN {X 0,Y 587.163,Z 160.707,A -85,B 0,C 180,E1 -1322.341,E2 -1322.341} C_VEL
LIN {X 0,Y 587.158,Z 156.87,A -85,B 0,C 180,E1 -1325.233,E2 -1325.233} C_VEL
LIN {X 0,Y 587.128,Z 153.068,A -85,B 0,C 180,E1 -1328.218,E2 -1328.218} C_VEL
LIN {X 0,Y 587.188,Z 149.641,A -85,B 0,C 180,E1 -1331.146,E2 -1331.146} C_VEL
LIN {X 0,Y 587.222,Z 146.127,A -85,B 0,C 180,E1 -1334.022,E2 -1334.022} C_VEL
LIN {X 0,Y 587.213,Z 143.568,A -85,B 0,C 180,E1 -1336.151,E2 -1336.151} C_VEL
LIN {X 0,Y 587.266,Z 140.196,A -85,B 0,C 180,E1 -1338.961,E2 -1338.961} C_VEL
LIN {X 0,Y 587.273,Z 139.35,A -85,B 0,C 180,E1 -1339.659,E2 -1339.659} C_VEL
LIN {X 0,Y 587.366,Z 139.322,A -85,B 0,C 180,E1 -1342.437,E2 -1342.437} C_VEL
LIN {X 0,Y 587.359,Z 139.325,A -85,B 0,C 180,E1 -1345.195,E2 -1345.195} C_VEL
LIN {X 0,Y 587.375,Z 139.32,A -85,B 0,C 180,E1 -1347.943,E2 -1347.943} C_VEL
LIN {X 0,Y 587.382,Z 139.319,A -85,B 0,C 180,E1 -1350.685,E2 -1350.685} C_VEL
LIN {X 0,Y 587.326,Z 139.328,A -85,B 0,C 180,E1 -1353.43,E2 -1353.43} C_VEL
LIN {X 0,Y 587.357,Z 139.322,A -85,B 0,C 180,E1 -1355.493,E2 -1355.493} C_VEL
LIN {X 0,Y 587.365,Z 139.323,A -85,B 0,C 180,E1 -1358.255,E2 -1358.255} C_VEL
LIN {X 0,Y 587.345,Z 139.325,A -85,B 0,C 180,E1 -1361.134,E2 -1361.134} C_VEL
LIN {X 0,Y 587.363,Z 139.323,A -85,B 0,C 180,E1 -1364.261,E2 -1364.261} C_VEL
LIN {X 0,Y 587.355,Z 139.322,A -85,B 0,C 180,E1 -1367.406,E2 -1367.406} C_VEL
LIN {X 0,Y 587.331,Z 139.327,A -85,B 0,C 180,E1 -1370.305,E2 -1370.305} C_VEL
LIN {X 0,Y 587.323,Z 139.327,A -85,B 0,C 180,E1 -1373.259,E2 -1373.259} C_VEL
LIN {X 0,Y 587.329,Z 139.327,A -85,B 0,C 180,E1 -1375.517,E2 -1375.517} C_VEL
LIN {X 0,Y 587.345,Z 139.326,A -85,B 0,C 180,E1 -1377.818,E2 -1377.818} C_VEL
LIN {X 0,Y 587.343,Z 139.324,A -85,B 0,C 180,E1 -1380.512,E2 -1380.512} C_VEL
LIN {X 0,Y 587.334,Z 139.326,A -85,B 0,C 180,E1 -1383.397,E2 -1383.397} C_VEL
LIN {X 0,Y 587.289,Z 139.332,A -85,B 0,C 180,E1 -1385.9,E2 -1385.9} C_VEL
LIN {X 0,Y 587.329,Z 139.328,A -85,B 0,C 180,E1 -1388.479,E2 -1388.479} C_VEL
LIN {X 0,Y 587.334,Z 139.327,A -85,B 0,C 180,E1 -1391.157,E2 -1391.157} C_VEL
LIN {X 0,Y 587.324,Z 139.326,A -85,B 0,C 180,E1 -1394.114,E2 -1394.114} C_VEL
LIN {X 0,Y 587.311,Z 139.331,A -85,B 0,C 180,E1 -1396.994,E2 -1396.994} C_VEL
LIN {X 0,Y 587.312,Z 139.329,A -85,B 0,C 180,E1 -1399.746,E2 -1399.746} C_VEL
LIN {X 0,Y 587.346,Z 139.323,A -85,B 0,C 180,E1 -1402.393,E2 -1402.393} C_VEL
LIN {X 0,Y 587.334,Z 139.325,A -85,B 0,C 180,E1 -1404.945,E2 -1404.945} C_VEL
LIN {X 0,Y 587.336,Z 139.325,A -85,B 0,C 180,E1 -1407.421,E2 -1407.421} C_VEL
LIN {X 0,Y 587.319,Z 139.327,A -85,B 0,C 180,E1 -1409.829,E2 -1409.829} C_VEL
LIN {X 0,Y 587.351,Z 139.323,A -85,B 0,C 180,E1 -1412.307,E2 -1412.307} C_VEL
LIN {X 0,Y 587.352,Z 139.325,A -85,B 0,C 180,E1 -1415.242,E2 -1415.242} C_VEL
LIN {X 0,Y 587.325,Z 139.326,A -85,B 0,C 180,E1 -1418.226,E2 -1418.226} C_VEL
LIN {X 0,Y 587.347,Z 139.327,A -85,B 0,C 180,E1 -1421.152,E2 -1421.152} C_VEL
LIN {X 0,Y 587.326,Z 139.326,A -85,B 0,C 180,E1 -1424.025,E2 -1424.025} C_VEL
LIN {X 0,Y 587.317,Z 139.328,A -85,B 0,C 180,E1 -1426.859,E2 -1426.859} C_VEL
LIN {X 0,Y 587.343,Z 139.327,A -85,B 0,C 180,E1 -1429.661,E2 -1429.661} C_VEL
LIN {X 0,Y 587.349,Z 139.324,A -85,B 0,C 180,E1 -1432.437,E2 -1432.437} C_VEL
LIN {X 0,Y 587.356,Z 139.322,A -85,B 0,C 180,E1 -1435.196,E2 -1435.196} C_VEL
LIN {X 0,Y 587.374,Z 139.322,A -85,B 0,C 180,E1 -1437.943,E2 -1437.943} C_VEL
LIN {X 0,Y 587.391,Z 139.32,A -85,B 0,C 180,E1 -1440.686,E2 -1440.686} C_VEL
LIN {X 0,Y 587.33,Z 139.326,A -85,B 0,C 180,E1 -1443.43,E2 -1443.43} C_VEL
LIN {X 0,Y 587.332,Z 139.326,A -85,B 0,C 180,E1 -1446.183,E2 -1446.183} C_VEL
LIN {X 0,Y 587.327,Z 139.329,A -85,B 0,C 180,E1 -1448.95,E2 -1448.95} C_VEL
LIN {X 0,Y 587.344,Z 139.324,A -85,B 0,C 180,E1 -1451.737,E2 -1451.737} C_VEL
LIN {X 0,Y 587.336,Z 139.325,A -85,B 0,C 180,E1 -1454.554,E2 -1454.554} C_VEL
LIN {X 0,Y 587.345,Z 139.327,A -85,B 0,C 180,E1 -1457.406,E2 -1457.406} C_VEL
LIN {X 0,Y 587.314,Z 139.329,A -85,B 0,C 180,E1 -1459.576,E2 -1459.576} C_VEL
LIN {X 0,Y 587.34,Z 139.325,A -85,B 0,C 180,E1 -1462.514,E2 -1462.514} C_VEL
LIN {X 0,Y 587.337,Z 139.325,A -85,B 0,C 180,E1 -1465.517,E2 -1465.517} C_VEL
LIN {X 0,Y 587.35,Z 139.323,A -85,B 0,C 180,E1 -1467.818,E2 -1467.818} C_VEL
LIN {X 0,Y 587.329,Z 139.327,A -85,B 0,C 180,E1 -1470.508,E2 -1470.508} C_VEL
LIN {X 0,Y 587.337,Z 139.328,A -85,B 0,C 180,E1 -1473.111,E2 -1473.111} C_VEL
LIN {X 0,Y 587.293,Z 139.33,A -85,B 0,C 180,E1 -1475.9,E2 -1475.9} C_VEL
LIN {X 0,Y 587.325,Z 139.326,A -85,B 0,C 180,E1 -1478.48,E2 -1478.48} C_VEL
LIN {X 0,Y 587.339,Z 139.325,A -85,B 0,C 180,E1 -1481.157,E2 -1481.157} C_VEL
LIN {X 0,Y 587.33,Z 139.327,A -85,B 0,C 180,E1 -1484.114,E2 -1484.114} C_VEL
LIN {X 0,Y 587.319,Z 139.326,A -85,B 0,C 180,E1 -1486.994,E2 -1486.994} C_VEL
LIN {X 0,Y 587.319,Z 139.328,A -85,B 0,C 180,E1 -1489.746,E2 -1489.746} C_VEL
LIN {X 0,Y 587.345,Z 139.327,A -85,B 0,C 180,E1 -1492.392,E2 -1492.392} C_VEL
LIN {X 0,Y 587.347,Z 139.463,A -85,B 0,C 180,E1 -1493.733,E2 -1493.733} C_VEL
LIN {X 0,Y 587.662,Z 143.269,A -85,B 0,C 180,E1 -1494.967,E2 -1494.967} C_VEL
LIN {X 0,Y 587.653,Z 149.27,A -85,B 0,C 180,E1 -1496.842,E2 -1496.842} C_VEL
LIN {X 0,Y 587.545,Z 157.871,A -85,B 0,C 180,E1 -1499.456,E2 -1499.456} C_VEL
LIN {X 0,Y 587.53,Z 167.383,A -85,B 0,C 180,E1 -1502.275,E2 -1502.275} C_VEL
LIN {X 0,Y 587.451,Z 177.69,A -85,B 0,C 180,E1 -1505.246,E2 -1505.246} C_VEL
LIN {X 0,Y 587.388,Z 188.282,A -85,B 0,C 180,E1 -1508.228,E2 -1508.228} C_VEL
LIN {X 0,Y 587.313,Z 198.873,A -85,B 0,C 180,E1 -1511.15,E2 -1511.15} C_VEL
LIN {X 0,Y 587.257,Z 209.464,A -85,B 0,C 180,E1 -1514.023,E2 -1514.023} C_VEL
LIN {X 0,Y 587.234,Z 220.055,A -85,B 0,C 180,E1 -1516.857,E2 -1516.857} C_VEL
LIN {X 0,Y 587.198,Z 223.572,A -85,B 0,C 180,E1 -1517.789,E2 -1517.789} C_VEL
LIN {X 0,Y 587.74,Z 228.092,A -85,B 0,C 180,E1 -1517.877,E2 -1517.877} C_VEL
LIN {X 0,Y 587.672,Z 241.739,A -85,B 0,C 180,E1 -1518.204,E2 -1518.204} C_VEL
LIN {X 0,Y 587.564,Z 254.425,A -85,B 0,C 180,E1 -1518.657,E2 -1518.657} C_VEL
LIN {X 0,Y 587.477,Z 266.21,A -85,B 0,C 180,E1 -1519.227,E2 -1519.227} C_VEL
LIN {X 0,Y 587.462,Z 277.477,A -85,B 0,C 180,E1 -1519.924,E2 -1519.924} C_VEL
LIN {X 0,Y 587.384,Z 287.648,A -85,B 0,C 180,E1 -1520.705,E2 -1520.705} C_VEL
LIN {X 0,Y 587.34,Z 296.788,A -85,B 0,C 180,E1 -1521.571,E2 -1521.571} C_VEL
LIN {X 0,Y 587.259,Z 305.692,A -85,B 0,C 180,E1 -1522.608,E2 -1522.608} C_VEL
LIN {X 0,Y 587.195,Z 312.747,A -85,B 0,C 180,E1 -1523.627,E2 -1523.627} C_VEL
LIN {X 0,Y 587.211,Z 317.681,A -85,B 0,C 180,E1 -1524.506,E2 -1524.506} C_VEL
LIN {X 0,Y 587.188,Z 322.372,A -85,B 0,C 180,E1 -1525.538,E2 -1525.538} C_VEL
LIN {X 0,Y 587.193,Z 325.956,A -85,B 0,C 180,E1 -1526.569,E2 -1526.569} C_VEL
LIN {X 0,Y 587.132,Z 327.809,A -85,B 0,C 180,E1 -1527.256,E2 -1527.256} C_VEL
LIN {X 0,Y 587.141,Z 329.202,A -85,B 0,C 180,E1 -1527.942,E2 -1527.942} C_VEL
LIN {X 0,Y 587.14,Z 330.784,A -85,B 0,C 180,E1 -1529.314,E2 -1529.314} C_VEL
LIN {X 0,Y 587.137,Z 331,A -85,B 0,C 180,E1 -1530,E2 -1530} C_VEL
LIN {X 0,Y 587.147,Z 330.184,A -85,B 0,C 180,E1 -1531.372,E2 -1531.372} C_VEL
LIN {X 0,Y 587.141,Z 329.202,A -85,B 0,C 180,E1 -1532.058,E2 -1532.058} C_VEL
LIN {X 0,Y 587.132,Z 327.809,A -85,B 0,C 180,E1 -1532.745,E2 -1532.745} C_VEL
LIN {X 0,Y 587.213,Z 324.896,A -85,B 0,C 180,E1 -1533.774,E2 -1533.774} C_VEL
LIN {X 0,Y 587.147,Z 320.949,A -85,B 0,C 180,E1 -1534.806,E2 -1534.806} C_VEL
LIN {X 0,Y 587.218,Z 314.876,A -85,B 0,C 180,E1 -1536.011,E2 -1536.011} C_VEL
LIN {X 0,Y 587.245,Z 308.235,A -85,B 0,C 180,E1 -1537.046,E2 -1537.046} C_VEL
LIN {X 0,Y 587.3,Z 299.988,A -85,B 0,C 180,E1 -1538.083,E2 -1538.083} C_VEL
LIN {X 0,Y 587.343,Z 291.535,A -85,B 0,C 180,E1 -1538.949,E2 -1538.949} C_VEL
LIN {X 0,Y 587.416,Z 281.09,A -85,B 0,C 180,E1 -1539.817,E2 -1539.817} C_VEL
LIN {X 0,Y 587.472,Z 270.755,A -85,B 0,C 180,E1 -1540.512,E2 -1540.512} C_VEL
LIN {X 0,Y 587.53,Z 259.161,A -85,B 0,C 180,E1 -1541.133,E2 -1541.133} C_VEL
LIN {X 0,Y 587.594,Z 246.69,A -85,B 0,C 180,E1 -1541.637,E2 -1541.637} C_VEL
LIN {X 0,Y 587.713,Z 233.431,A -85,B 0,C 180,E1 -1542.014,E2 -1542.014} C_VEL
LIN {X 0,Y 587.492,Z 225.602,A -85,B 0,C 180,E1 -1542.172,E2 -1542.172} C_VEL
LIN {X 0,Y 587.197,Z 223.53,A -85,B 0,C 180,E1 -1542.222,E2 -1542.222} C_VEL
LIN {X 0,Y 587.256,Z 213.435,A -85,B 0,C 180,E1 -1544.91,E2 -1544.91} C_VEL
LIN {X 0,Y 587.303,Z 202.844,A -85,B 0,C 180,E1 -1547.767,E2 -1547.767} C_VEL
LIN {X 0,Y 587.378,Z 192.252,A -85,B 0,C 180,E1 -1550.669,E2 -1550.669} C_VEL
LIN {X 0,Y 587.436,Z 181.661,A -85,B 0,C 180,E1 -1553.628,E2 -1553.628} C_VEL
LIN {X 0,Y 587.489,Z 172.394,A -85,B 0,C 180,E1 -1556.272,E2 -1556.272} C_VEL
LIN {X 0,Y 587.484,Z 164.45,A -85,B 0,C 180,E1 -1558.589,E2 -1558.589} C_VEL
LIN {X 0,Y 587.616,Z 155.183,A -85,B 0,C 180,E1 -1561.35,E2 -1561.35} C_VEL
LIN {X 0,Y 587.648,Z 147.24,A -85,B 0,C 180,E1 -1563.788,E2 -1563.788} C_VEL
LIN {X 0,Y 587.552,Z 140.62,A -85,B 0,C 180,E1 -1565.882,E2 -1565.882} C_VEL
LIN {X 0,Y 587.315,Z 139.331,A -85,B 0,C 180,E1 -1566.323,E2 -1566.323} C_VEL
LIN {X 0,Y 587.329,Z 139.328,A -85,B 0,C 180,E1 -1568.941,E2 -1568.941} C_VEL
LIN {X 0,Y 587.358,Z 139.325,A -85,B 0,C 180,E1 -1572.072,E2 -1572.072} C_VEL
LIN {X 0,Y 587.321,Z 139.329,A -85,B 0,C 180,E1 -1575.089,E2 -1575.089} C_VEL
LIN {X 0,Y 587.327,Z 139.328,A -85,B 0,C 180,E1 -1577.925,E2 -1577.925} C_VEL
LIN {X 0,Y 587.35,Z 139.325,A -85,B 0,C 180,E1 -1580.641,E2 -1580.641} C_VEL
LIN {X 0,Y 587.353,Z 139.326,A -85,B 0,C 180,E1 -1583.292,E2 -1583.292} C_VEL
LIN {X 0,Y 587.37,Z 139.322,A -85,B 0,C 180,E1 -1585.78,E2 -1585.78} C_VEL
LIN {X 0,Y 587.35,Z 139.326,A -85,B 0,C 180,E1 -1588.231,E2 -1588.231} C_VEL
LIN {X 0,Y 587.355,Z 139.323,A -85,B 0,C 180,E1 -1590.866,E2 -1590.866} C_VEL
LIN {X 0,Y 587.364,Z 139.323,A -85,B 0,C 180,E1 -1593.819,E2 -1593.819} C_VEL
LIN {X 0,Y 587.329,Z 139.327,A -85,B 0,C 180,E1 -1595.993,E2 -1595.993} C_VEL
LIN {X 0,Y 587.324,Z 139.328,A -85,B 0,C 180,E1 -1598.225,E2 -1598.225} C_VEL
LIN {X 0,Y 587.354,Z 139.324,A -85,B 0,C 180,E1 -1601.151,E2 -1601.151} C_VEL
LIN {X 0,Y 587.324,Z 139.327,A -85,B 0,C 180,E1 -1604.024,E2 -1604.024} C_VEL
LIN {X 0,Y 587.363,Z 139.323,A -85,B 0,C 180,E1 -1606.154,E2 -1606.154} C_VEL
LIN {X 0,Y 587.344,Z 139.325,A -85,B 0,C 180,E1 -1608.962,E2 -1608.962} C_VEL
LIN {X 0,Y 587.37,Z 139.323,A -85,B 0,C 180,E1 -1611.744,E2 -1611.744} C_VEL
LIN {X 0,Y 587.363,Z 139.324,A -85,B 0,C 180,E1 -1614.507,E2 -1614.507} C_VEL
LIN {X 0,Y 587.374,Z 139.321,A -85,B 0,C 180,E1 -1617.256,E2 -1617.256} C_VEL
LIN {X 0,Y 587.389,Z 139.32,A -85,B 0,C 180,E1 -1620,E2 -1620} C_VEL
LIN {X 0,Y 587.377,Z 139.323,A -85,B 0,C 180,E1 -1622.743,E2 -1622.743} C_VEL
LIN {X 0,Y 587.355,Z 139.325,A -85,B 0,C 180,E1 -1625.493,E2 -1625.493} C_VEL
LIN {X 0,Y 587.367,Z 139.322,A -85,B 0,C 180,E1 -1628.255,E2 -1628.255} C_VEL
LIN {X 0,Y 587.275,Z 139.459,A -85,B 0,C 180,E1 -1630.341,E2 -1630.341} C_VEL
LIN {X 0,Y 587.221,Z 142.88,A -85,B 0,C 180,E1 -1633.143,E2 -1633.143} C_VEL
LIN {X 0,Y 587.22,Z 145.407,A -85,B 0,C 180,E1 -1635.266,E2 -1635.266} C_VEL
LIN {X 0,Y 587.22,Z 147.954,A -85,B 0,C 180,E1 -1637.41,E2 -1637.41} C_VEL
LIN {X 0,Y 587.181,Z 148.939,A -85,B 0,C 180,E1 -1638.232,E2 -1638.232} C_VEL
LIN {X 0,Y 586.506,Z 149.693,A -85,B 0,C 180,E1 -1638.8,E2 -1638.8} C_VEL
LIN {X 0,Y 583.644,Z 151.085,A -85,B 0,C 180,E1 -1639.718,E2 -1639.718} C_VEL
LIN {X 0,Y 581.225,Z 152.184,A -85,B 0,C 180,E1 -1640.458,E2 -1640.458} C_VEL
LIN {X 0,Y 580.176,Z 152.92,A -85,B 0,C 180,E1 -1641.03,E2 -1641.03} C_VEL
LIN {X 0,Y 580.086,Z 153.136,A -85,B 0,C 180,E1 -1641.224,E2 -1641.224} C_VEL
LIN {X 0,Y 580.078,Z 156.515,A -85,B 0,C 180,E1 -1644.326,E2 -1644.326} C_VEL
LIN {X 0,Y 580.066,Z 160.551,A -85,B 0,C 180,E1 -1647.413,E2 -1647.413} C_VEL
LIN {X 0,Y 580.049,Z 163.703,A -85,B 0,C 180,E1 -1649.786,E2 -1649.786} C_VEL
LIN {X 0,Y 580.067,Z 167.835,A -85,B 0,C 180,E1 -1652.755,E2 -1652.755} C_VEL
LIN {X 0,Y 580.779,Z 174.14,A -85,B 0,C 180,E1 -1652.903,E2 -1652.903} C_VEL
LIN {X 0,Y 580.673,Z 187.541,A -85,B 0,C 180,E1 -1653.297,E2 -1653.297} C_VEL
LIN {X 0,Y 580.563,Z 199.047,A -85,B 0,C 180,E1 -1653.771,E2 -1653.771} C_VEL
LIN {X 0,Y 580.454,Z 210.174,A -85,B 0,C 180,E1 -1654.369,E2 -1654.369} C_VEL
LIN {X 0,Y 580.42,Z 221.106,A -85,B 0,C 180,E1 -1655.11,E2 -1655.11} C_VEL
LIN {X 0,Y 580.344,Z 230.392,A -85,B 0,C 180,E1 -1655.883,E2 -1655.883} C_VEL
LIN {X 0,Y 580.242,Z 239.386,A -85,B 0,C 180,E1 -1656.793,E2 -1656.793} C_VEL
LIN {X 0,Y 580.167,Z 247.888,A -85,B 0,C 180,E1 -1657.863,E2 -1657.863} C_VEL
LIN {X 0,Y 580.137,Z 255.37,A -85,B 0,C 180,E1 -1659.046,E2 -1659.046} C_VEL
LIN {X 0,Y 580.119,Z 261.234,A -85,B 0,C 180,E1 -1660.25,E2 -1660.25} C_VEL
LIN {X 0,Y 580.047,Z 265.143,A -85,B 0,C 180,E1 -1661.304,E2 -1661.304} C_VEL
LIN {X 0,Y 580.081,Z 267.99,A -85,B 0,C 180,E1 -1662.349,E2 -1662.349} C_VEL
LIN {X 0,Y 580.026,Z 270.214,A -85,B 0,C 180,E1 -1663.681,E2 -1663.681} C_VEL
LIN {X 0,Y 580.034,Z 270.917,A -85,B 0,C 180,E1 -1664.648,E2 -1664.648} C_VEL
LIN {X 0,Y 580.038,Z 270.856,A -85,B 0,C 180,E1 -1665.632,E2 -1665.632} C_VEL
LIN {X 0,Y 580.03,Z 269.954,A -85,B 0,C 180,E1 -1666.635,E2 -1666.635} C_VEL
LIN {X 0,Y 580.063,Z 268.175,A -85,B 0,C 180,E1 -1667.652,E2 -1667.652} C_VEL
LIN {X 0,Y 580.073,Z 265.429,A -85,B 0,C 180,E1 -1668.692,E2 -1668.692} C_VEL
LIN {X 0,Y 580.118,Z 261.606,A -85,B 0,C 180,E1 -1669.749,E2 -1669.749} C_VEL
LIN {X 0,Y 580.137,Z 255.877,A -85,B 0,C 180,E1 -1670.953,E2 -1670.953} C_VEL
LIN {X 0,Y 580.168,Z 248.53,A -85,B 0,C 180,E1 -1672.136,E2 -1672.136} C_VEL
LIN {X 0,Y 580.24,Z 240.173,A -85,B 0,C 180,E1 -1673.206,E2 -1673.206} C_VEL
LIN {X 0,Y 580.336,Z 231.385,A -85,B 0,C 180,E1 -1674.117,E2 -1674.117} C_VEL
LIN {X 0,Y 580.429,Z 220.895,A -85,B 0,C 180,E1 -1674.996,E2 -1674.996} C_VEL
LIN {X 0,Y 580.457,Z 209.94,A -85,B 0,C 180,E1 -1675.736,E2 -1675.736} C_VEL
LIN {X 0,Y 580.552,Z 198.1,A -85,B 0,C 180,E1 -1676.363,E2 -1676.363} C_VEL
LIN {X 0,Y 580.677,Z 186.58,A -85,B 0,C 180,E1 -1676.826,E2 -1676.826} C_VEL
LIN {X 0,Y 580.785,Z 173.077,A -85,B 0,C 180,E1 -1677.213,E2 -1677.213} C_VEL
LIN {X 0,Y 580.051,Z 167.679,A -85,B 0,C 180,E1 -1677.347,E2 -1677.347} C_VEL
LIN {X 0,Y 580.044,Z 163.824,A -85,B 0,C 180,E1 -1680.213,E2 -1680.213} C_VEL
LIN {X 0,Y 580.064,Z 160.671,A -85,B 0,C 180,E1 -1682.587,E2 -1682.587} C_VEL
LIN {X 0,Y 580.068,Z 157.087,A -85,B 0,C 180,E1 -1685.323,E2 -1685.323} C_VEL
LIN {X 0,Y 580.062,Z 153.993,A -85,B 0,C 180,E1 -1687.939,E2 -1687.939} C_VEL
LIN {X 0,Y 580.074,Z 151.394,A -85,B 0,C 180,E1 -1690.169,E2 -1690.169} C_VEL
LIN {X 0,Y 580.138,Z 147.765,A -85,B 0,C 180,E1 -1693.142,E2 -1693.142} C_VEL
LIN {X 0,Y 580.168,Z 144.39,A -85,B 0,C 180,E1 -1695.979,E2 -1695.979} C_VEL
LIN {X 0,Y 580.206,Z 140.95,A -85,B 0,C 180,E1 -1698.854,E2 -1698.854} C_VEL
LIN {X 0,Y 580.214,Z 140.215,A -85,B 0,C 180,E1 -1699.532,E2 -1699.532} C_VEL
LIN {X 0,Y 580.327,Z 140.198,A -85,B 0,C 180,E1 -1702.344,E2 -1702.344} C_VEL
LIN {X 0,Y 580.331,Z 140.2,A -85,B 0,C 180,E1 -1705.137,E2 -1705.137} C_VEL
LIN {X 0,Y 580.344,Z 140.196,A -85,B 0,C 180,E1 -1707.918,E2 -1707.918} C_VEL
LIN {X 0,Y 580.353,Z 140.195,A -85,B 0,C 180,E1 -1710.694,E2 -1710.694} C_VEL
LIN {X 0,Y 580.279,Z 140.206,A -85,B 0,C 180,E1 -1713.472,E2 -1713.472} C_VEL
LIN {X 0,Y 580.323,Z 140.198,A -85,B 0,C 180,E1 -1715.56,E2 -1715.56} C_VEL
LIN {X 0,Y 580.327,Z 140.201,A -85,B 0,C 180,E1 -1718.356,E2 -1718.356} C_VEL
LIN {X 0,Y 580.297,Z 140.202,A -85,B 0,C 180,E1 -1721.191,E2 -1721.191} C_VEL
LIN {X 0,Y 580.326,Z 140.198,A -85,B 0,C 180,E1 -1724.017,E2 -1724.017} C_VEL
LIN {X 0,Y 580.309,Z 140.203,A -85,B 0,C 180,E1 -1726.914,E2 -1726.914} C_VEL
LIN {X 0,Y 580.304,Z 140.201,A -85,B 0,C 180,E1 -1729.822,E2 -1729.822} C_VEL
LIN {X 0,Y 580.294,Z 140.205,A -85,B 0,C 180,E1 -1732.802,E2 -1732.802} C_VEL
LIN {X 0,Y 580.303,Z 140.202,A -85,B 0,C 180,E1 -1735.08,E2 -1735.08} C_VEL
LIN {X 0,Y 580.297,Z 140.201,A -85,B 0,C 180,E1 -1738.186,E2 -1738.186} C_VEL
LIN {X 0,Y 580.288,Z 140.203,A -85,B 0,C 180,E1 -1740.696,E2 -1740.696} C_VEL
LIN {X 0,Y 580.303,Z 140.201,A -85,B 0,C 180,E1 -1743.317,E2 -1743.317} C_VEL
LIN {X 0,Y 580.244,Z 140.209,A -85,B 0,C 180,E1 -1745.757,E2 -1745.757} C_VEL
LIN {X 0,Y 580.285,Z 140.203,A -85,B 0,C 180,E1 -1748.147,E2 -1748.147} C_VEL
LIN {X 0,Y 580.297,Z 140.203,A -85,B 0,C 180,E1 -1750.844,E2 -1750.844} C_VEL
LIN {X 0,Y 580.277,Z 140.205,A -85,B 0,C 180,E1 -1753.658,E2 -1753.658} C_VEL
LIN {X 0,Y 580.274,Z 140.205,A -85,B 0,C 180,E1 -1756.61,E2 -1756.61} C_VEL
LIN {X 0,Y 580.298,Z 140.203,A -85,B 0,C 180,E1 -1759.157,E2 -1759.157} C_VEL
LIN {X 0,Y 580.291,Z 140.205,A -85,B 0,C 180,E1 -1761.927,E2 -1761.927} C_VEL
LIN {X 0,Y 580.282,Z 140.206,A -85,B 0,C 180,E1 -1764.455,E2 -1764.455} C_VEL
LIN {X 0,Y 580.287,Z 140.204,A -85,B 0,C 180,E1 -1766.975,E2 -1766.975} C_VEL
LIN {X 0,Y 580.29,Z 140.203,A -85,B 0,C 180,E1 -1769.425,E2 -1769.425} C_VEL
LIN {X 0,Y 580.298,Z 140.201,A -85,B 0,C 180,E1 -1772.142,E2 -1772.142} C_VEL
LIN {X 0,Y 580.322,Z 140.201,A -85,B 0,C 180,E1 -1775.27,E2 -1775.27} C_VEL
LIN {X 0,Y 580.275,Z 140.205,A -85,B 0,C 180,E1 -1777.948,E2 -1777.948} C_VEL
LIN {X 0,Y 580.302,Z 140.202,A -85,B 0,C 180,E1 -1780.914,E2 -1780.914} C_VEL
LIN {X 0,Y 580.275,Z 140.206,A -85,B 0,C 180,E1 -1783.826,E2 -1783.826} C_VEL
LIN {X 0,Y 580.274,Z 140.205,A -85,B 0,C 180,E1 -1786.696,E2 -1786.696} C_VEL
LIN {X 0,Y 580.302,Z 140.203,A -85,B 0,C 180,E1 -1789.534,E2 -1789.534} C_VEL
LIN {X 0,Y 580.315,Z 140.2,A -85,B 0,C 180,E1 -1792.345,E2 -1792.345} C_VEL
LIN {X 0,Y 580.329,Z 140.197,A -85,B 0,C 180,E1 -1795.137,E2 -1795.137} C_VEL
LIN {X 0,Y 580.344,Z 140.198,A -85,B 0,C 180,E1 -1797.918,E2 -1797.918} C_VEL
LIN {X 0,Y 580.362,Z 140.195,A -85,B 0,C 180,E1 -1800.694,E2 -1800.694} C_VEL
LIN {X 0,Y 580.282,Z 140.203,A -85,B 0,C 180,E1 -1803.472,E2 -1803.472} C_VEL
LIN {X 0,Y 580.33,Z 140.199,A -85,B 0,C 180,E1 -1805.56,E2 -1805.56} C_VEL
LIN {X 0,Y 580.313,Z 140.2,A -85,B 0,C 180,E1 -1808.357,E2 -1808.357} C_VEL
LIN {X 0,Y 580.303,Z 140.202,A -85,B 0,C 180,E1 -1811.191,E2 -1811.191} C_VEL
LIN {X 0,Y 580.317,Z 140.201,A -85,B 0,C 180,E1 -1814.018,E2 -1814.018} C_VEL
LIN {X 0,Y 580.316,Z 140.199,A -85,B 0,C 180,E1 -1816.914,E2 -1816.914} C_VEL
LIN {X 0,Y 580.288,Z 140.206,A -85,B 0,C 180,E1 -1819.823,E2 -1819.823} C_VEL
LIN {X 0,Y 580.275,Z 140.206,A -85,B 0,C 180,E1 -1822.053,E2 -1822.053} C_VEL
LIN {X 0,Y 580.31,Z 140.2,A -85,B 0,C 180,E1 -1825.08,E2 -1825.08} C_VEL
LIN {X 0,Y 580.301,Z 140.204,A -85,B 0,C 180,E1 -1828.186,E2 -1828.186} C_VEL
LIN {X 0,Y 580.284,Z 140.206,A -85,B 0,C 180,E1 -1830.694,E2 -1830.694} C_VEL
LIN {X 0,Y 580.285,Z 140.205,A -85,B 0,C 180,E1 -1833.313,E2 -1833.313} C_VEL
LIN {X 0,Y 580.248,Z 140.209,A -85,B 0,C 180,E1 -1835.756,E2 -1835.756} C_VEL
LIN {X 0,Y 580.288,Z 140.204,A -85,B 0,C 180,E1 -1838.147,E2 -1838.147} C_VEL
LIN {X 0,Y 580.301,Z 140.201,A -85,B 0,C 180,E1 -1840.844,E2 -1840.844} C_VEL
LIN {X 0,Y 580.282,Z 140.204,A -85,B 0,C 180,E1 -1843.658,E2 -1843.658} C_VEL
LIN {X 0,Y 580.278,Z 140.205,A -85,B 0,C 180,E1 -1846.61,E2 -1846.61} C_VEL
LIN {X 0,Y 580.301,Z 140.202,A -85,B 0,C 180,E1 -1849.157,E2 -1849.157} C_VEL
LIN {X 0,Y 580.29,Z 140.204,A -85,B 0,C 180,E1 -1851.928,E2 -1851.928} C_VEL
LIN {X 0,Y 580.319,Z 140.33,A -85,B 0,C 180,E1 -1853.505,E2 -1853.505} C_VEL
LIN {X 0,Y 580.728,Z 144.593,A -85,B 0,C 180,E1 -1854.911,E2 -1854.911} C_VEL
LIN {X 0,Y 580.637,Z 152.536,A -85,B 0,C 180,E1 -1857.41,E2 -1857.41} C_VEL
LIN {X 0,Y 580.577,Z 161.803,A -85,B 0,C 180,E1 -1860.244,E2 -1860.244} C_VEL
LIN {X 0,Y 580.446,Z 171.071,A -85,B 0,C 180,E1 -1862.996,E2 -1862.996} C_VEL
LIN {X 0,Y 580.394,Z 180.338,A -85,B 0,C 180,E1 -1865.688,E2 -1865.688} C_VEL
LIN {X 0,Y 580.361,Z 189.605,A -85,B 0,C 180,E1 -1868.325,E2 -1868.325} C_VEL
LIN {X 0,Y 580.26,Z 200.197,A -85,B 0,C 180,E1 -1871.279,E2 -1871.279} C_VEL
LIN {X 0,Y 580.215,Z 209.464,A -85,B 0,C 180,E1 -1873.824,E2 -1873.824} C_VEL
LIN {X 0,Y 580.186,Z 220.055,A -85,B 0,C 180,E1 -1876.694,E2 -1876.694} C_VEL
LIN {X 0,Y 580.122,Z 223.53,A -85,B 0,C 180,E1 -1877.627,E2 -1877.627} C_VEL
LIN {X 0,Y 580.801,Z 229.234,A -85,B 0,C 180,E1 -1877.752,E2 -1877.752} C_VEL
LIN {X 0,Y 580.734,Z 242.499,A -85,B 0,C 180,E1 -1878.083,E2 -1878.083} C_VEL
LIN {X 0,Y 580.598,Z 254.637,A -85,B 0,C 180,E1 -1878.528,E2 -1878.528} C_VEL
LIN {X 0,Y 580.487,Z 266.211,A -85,B 0,C 180,E1 -1879.096,E2 -1879.096} C_VEL
LIN {X 0,Y 580.451,Z 277.478,A -85,B 0,C 180,E1 -1879.801,E2 -1879.801} C_VEL
LIN {X 0,Y 580.352,Z 287.648,A -85,B 0,C 180,E1 -1880.591,E2 -1880.591} C_VEL
LIN {X 0,Y 580.279,Z 296.788,A -85,B 0,C 180,E1 -1881.468,E2 -1881.468} C_VEL
LIN {X 0,Y 580.199,Z 305.692,A -85,B 0,C 180,E1 -1882.518,E2 -1882.518} C_VEL
LIN {X 0,Y 580.12,Z 312.467,A -85,B 0,C 180,E1 -1883.505,E2 -1883.505} C_VEL
LIN {X 0,Y 580.139,Z 317.681,A -85,B 0,C 180,E1 -1884.439,E2 -1884.439} C_VEL
LIN {X 0,Y 580.108,Z 322.372,A -85,B 0,C 180,E1 -1885.484,E2 -1885.484} C_VEL
LIN {X 0,Y 580.123,Z 325.957,A -85,B 0,C 180,E1 -1886.527,E2 -1886.527} C_VEL
LIN {X 0,Y 580.043,Z 327.809,A -85,B 0,C 180,E1 -1887.222,E2 -1887.222} C_VEL
LIN {X 0,Y 580.04,Z 329.201,A -85,B 0,C 180,E1 -1887.917,E2 -1887.917} C_VEL
LIN {X 0,Y 580.04,Z 330.784,A -85,B 0,C 180,E1 -1889.306,E2 -1889.306} C_VEL
LIN {X 0,Y 580.037,Z 331,A -85,B 0,C 180,E1 -1890,E2 -1890} C_VEL
LIN {X 0,Y 580.047,Z 330.185,A -85,B 0,C 180,E1 -1891.389,E2 -1891.389} C_VEL
LIN {X 0,Y 580.04,Z 329.201,A -85,B 0,C 180,E1 -1892.083,E2 -1892.083} C_VEL
LIN {X 0,Y 580.043,Z 327.809,A -85,B 0,C 180,E1 -1892.778,E2 -1892.778} C_VEL
LIN {X 0,Y 580.11,Z 324.896,A -85,B 0,C 180,E1 -1893.821,E2 -1893.821} C_VEL
LIN {X 0,Y 580.053,Z 320.949,A -85,B 0,C 180,E1 -1894.865,E2 -1894.865} C_VEL
LIN {X 0,Y 580.139,Z 314.877,A -85,B 0,C 180,E1 -1896.085,E2 -1896.085} C_VEL
LIN {X 0,Y 580.184,Z 308.235,A -85,B 0,C 180,E1 -1897.133,E2 -1897.133} C_VEL
LIN {X 0,Y 580.25,Z 299.988,A -85,B 0,C 180,E1 -1898.182,E2 -1898.182} C_VEL
LIN {X 0,Y 580.308,Z 291.535,A -85,B 0,C 180,E1 -1899.059,E2 -1899.059} C_VEL
LIN {X 0,Y 580.417,Z 281.091,A -85,B 0,C 180,E1 -1899.936,E2 -1899.936} C_VEL
LIN {X 0,Y 580.475,Z 270.756,A -85,B 0,C 180,E1 -1900.64,E2 -1900.64} C_VEL
LIN {X 0,Y 580.564,Z 259.59,A -85,B 0,C 180,E1 -1901.248,E2 -1901.248} C_VEL
LIN {X 0,Y 580.635,Z 247.762,A -85,B 0,C 180,E1 -1901.742,E2 -1901.742} C_VEL
LIN {X 0,Y 580.766,Z 234.344,A -85,B 0,C 180,E1 -1902.138,E2 -1902.138} C_VEL
LIN {X 0,Y 580.592,Z 226.484,A -85,B 0,C 180,E1 -1902.305,E2 -1902.305} C_VEL
LIN {X 0,Y 580.122,Z 223.53,A -85,B 0,C 180,E1 -1902.373,E2 -1902.373} C_VEL
LIN {X 0,Y 580.217,Z 213.435,A -85,B 0,C 180,E1 -1905.095,E2 -1905.095} C_VEL
LIN {X 0,Y 580.252,Z 202.844,A -85,B 0,C 180,E1 -1907.99,E2 -1907.99} C_VEL
LIN {X 0,Y 580.345,Z 192.49,A -85,B 0,C 180,E1 -1910.865,E2 -1910.865} C_VEL
LIN {X 0,Y 580.407,Z 182.985,A -85,B 0,C 180,E1 -1913.553,E2 -1913.553} C_VEL
LIN {X 0,Y 580.484,Z 173.22,A -85,B 0,C 180,E1 -1916.372,E2 -1916.372} C_VEL
LIN {X 0,Y 580.507,Z 164.45,A -85,B 0,C 180,E1 -1918.965,E2 -1918.965} C_VEL
LIN {X 0,Y 580.652,Z 155.343,A -85,B 0,C 180,E1 -1921.721,E2 -1921.721} C_VEL
LIN {X 0,Y 580.707,Z 147.32,A -85,B 0,C 180,E1 -1924.222,E2 -1924.222} C_VEL
LIN {X 0,Y 580.644,Z 142.367,A -85,B 0,C 180,E1 -1925.81,E2 -1925.81} C_VEL
LIN {X 0,Y 580.307,Z 140.204,A -85,B 0,C 180,E1 -1926.591,E2 -1926.591} C_VEL
LIN {X 0,Y 580.301,Z 140.205,A -85,B 0,C 180,E1 -1929.185,E2 -1929.185} C_VEL
LIN {X 0,Y 580.303,Z 140.202,A -85,B 0,C 180,E1 -1931.767,E2 -1931.767} C_VEL
LIN {X 0,Y 580.272,Z 140.206,A -85,B 0,C 180,E1 -1934.626,E2 -1934.626} C_VEL
LIN {X 0,Y 580.291,Z 140.204,A -85,B 0,C 180,E1 -1937.628,E2 -1937.628} C_VEL
LIN {X 0,Y 580.299,Z 140.204,A -85,B 0,C 180,E1 -1940.067,E2 -1940.067} C_VEL
LIN {X 0,Y 580.303,Z 140.203,A -85,B 0,C 180,E1 -1943.066,E2 -1943.066} C_VEL
LIN {X 0,Y 580.323,Z 140.2,A -85,B 0,C 180,E1 -1946.145,E2 -1946.145} C_VEL
LIN {X 0,Y 580.286,Z 140.205,A -85,B 0,C 180,E1 -1948.615,E2 -1948.615} C_VEL
LIN {X 0,Y 580.297,Z 140.203,A -85,B 0,C 180,E1 -1951.024,E2 -1951.024} C_VEL
LIN {X 0,Y 580.296,Z 140.204,A -85,B 0,C 180,E1 -1953.666,E2 -1953.666} C_VEL
LIN {X 0,Y 580.301,Z 140.203,A -85,B 0,C 180,E1 -1955.683,E2 -1955.683} C_VEL
LIN {X 0,Y 580.275,Z 140.205,A -85,B 0,C 180,E1 -1957.947,E2 -1957.947} C_VEL
LIN {X 0,Y 580.304,Z 140.202,A -85,B 0,C 180,E1 -1960.913,E2 -1960.913} C_VEL
LIN {X 0,Y 580.275,Z 140.206,A -85,B 0,C 180,E1 -1963.825,E2 -1963.825} C_VEL
LIN {X 0,Y 580.331,Z 140.198,A -85,B 0,C 180,E1 -1965.983,E2 -1965.983} C_VEL
LIN {X 0,Y 580.31,Z 140.202,A -85,B 0,C 180,E1 -1968.827,E2 -1968.827} C_VEL
LIN {X 0,Y 580.333,Z 140.2,A -85,B 0,C 180,E1 -1971.644,E2 -1971.644} C_VEL
LIN {X 0,Y 580.329,Z 140.2,A -85,B 0,C 180,E1 -1974.44,E2 -1974.44} C_VEL
LIN {X 0,Y 580.341,Z 140.197,A -85,B 0,C 180,E1 -1977.223,E2 -1977.223} C_VEL
LIN {X 0,Y 580.359,Z 140.195,A -85,B 0,C 180,E1 -1980,E2 -1980} C_VEL
LIN {X 0,Y 580.343,Z 140.199,A -85,B 0,C 180,E1 -1982.776,E2 -1982.776} C_VEL
LIN {X 0,Y 580.322,Z 140.201,A -85,B 0,C 180,E1 -1985.559,E2 -1985.559} C_VEL
LIN {X 0,Y 580.329,Z 140.199,A -85,B 0,C 180,E1 -1988.356,E2 -1988.356} C_VEL
LIN {X 0,Y 580.217,Z 140.3,A -85,B 0,C 180,E1 -1990.468,E2 -1990.468} C_VEL
LIN {X 0,Y 580.162,Z 143.756,A -85,B 0,C 180,E1 -1993.306,E2 -1993.306} C_VEL
LIN {X 0,Y 580.169,Z 147.149,A -85,B 0,C 180,E1 -1996.177,E2 -1996.177} C_VEL
LIN {X 0,Y 580.125,Z 150.588,A -85,B 0,C 180,E1 -1999.1,E2 -1999.1} C_VEL
LIN {X 0,Y 580.086,Z 153.136,A -85,B 0,C 180,E1 -2001.224,E2 -2001.224} C_VEL
LIN {X 0,Y 579.396,Z 153.817,A -85,B 0,C 180,E1 -2001.799,E2 -2001.799} C_VEL
LIN {X 0,Y 576.503,Z 155.106,A -85,B 0,C 180,E1 -2002.731,E2 -2002.731} C_VEL
LIN {X 0,Y 574.077,Z 156.156,A -85,B 0,C 180,E1 -2003.481,E2 -2003.481} C_VEL
LIN {X 0,Y 573.049,Z 156.888,A -85,B 0,C 180,E1 -2004.06,E2 -2004.06} C_VEL
LIN {X 0,Y 572.973,Z 157.111,A -85,B 0,C 180,E1 -2004.257,E2 -2004.257} C_VEL
LIN {X 0,Y 572.96,Z 160.296,A -85,B 0,C 180,E1 -2006.99,E2 -2006.99} C_VEL
LIN {X 0,Y 572.971,Z 163.5,A -85,B 0,C 180,E1 -2009.439,E2 -2009.439} C_VEL
LIN {X 0,Y 572.941,Z 167.385,A -85,B 0,C 180,E1 -2012.368,E2 -2012.368} C_VEL
LIN {X 0,Y 572.942,Z 167.682,A -85,B 0,C 180,E1 -2012.59,E2 -2012.59} C_VEL
LIN {X 0,Y 573.823,Z 174.595,A -85,B 0,C 180,E1 -2012.764,E2 -2012.764} C_VEL
LIN {X 0,Y 573.723,Z 187.098,A -85,B 0,C 180,E1 -2013.137,E2 -2013.137} C_VEL
LIN {X 0,Y 573.592,Z 199.234,A -85,B 0,C 180,E1 -2013.641,E2 -2013.641} C_VEL
LIN {X 0,Y 573.443,Z 211.441,A -85,B 0,C 180,E1 -2014.316,E2 -2014.316} C_VEL
LIN {X 0,Y 573.387,Z 222.121,A -85,B 0,C 180,E1 -2015.064,E2 -2015.064} C_VEL
LIN {X 0,Y 573.296,Z 230.726,A -85,B 0,C 180,E1 -2015.8,E2 -2015.8} C_VEL
LIN {X 0,Y 573.187,Z 239.531,A -85,B 0,C 180,E1 -2016.707,E2 -2016.707} C_VEL
LIN {X 0,Y 573.105,Z 248.189,A -85,B 0,C 180,E1 -2017.817,E2 -2017.817} C_VEL
LIN {X 0,Y 573.077,Z 253.903,A -85,B 0,C 180,E1 -2018.714,E2 -2018.714} C_VEL
LIN {X 0,Y 573.053,Z 258.703,A -85,B 0,C 180,E1 -2019.623,E2 -2019.623} C_VEL
LIN {X 0,Y 573.008,Z 262.664,A -85,B 0,C 180,E1 -2020.545,E2 -2020.545} C_VEL
LIN {X 0,Y 573.004,Z 267.141,A -85,B 0,C 180,E1 -2021.965,E2 -2021.965} C_VEL
LIN {X 0,Y 572.973,Z 268.598,A -85,B 0,C 180,E1 -2022.612,E2 -2022.612} C_VEL
LIN {X 0,Y 572.926,Z 270.181,A -85,B 0,C 180,E1 -2023.635,E2 -2023.635} C_VEL
LIN {X 0,Y 572.935,Z 270.917,A -85,B 0,C 180,E1 -2024.645,E2 -2024.645} C_VEL
LIN {X 0,Y 572.938,Z 270.858,A -85,B 0,C 180,E1 -2025.637,E2 -2025.637} C_VEL
LIN {X 0,Y 572.933,Z 270.002,A -85,B 0,C 180,E1 -2026.612,E2 -2026.612} C_VEL
LIN {X 0,Y 572.985,Z 268.396,A -85,B 0,C 180,E1 -2027.576,E2 -2027.576} C_VEL
LIN {X 0,Y 573.001,Z 266.073,A -85,B 0,C 180,E1 -2028.522,E2 -2028.522} C_VEL
LIN {X 0,Y 573.009,Z 262.835,A -85,B 0,C 180,E1 -2029.502,E2 -2029.502} C_VEL
LIN {X 0,Y 573.051,Z 258.113,A -85,B 0,C 180,E1 -2030.591,E2 -2030.591} C_VEL
LIN {X 0,Y 573.097,Z 251.925,A -85,B 0,C 180,E1 -2031.706,E2 -2031.706} C_VEL
LIN {X 0,Y 573.158,Z 243.957,A -85,B 0,C 180,E1 -2032.846,E2 -2032.846} C_VEL
LIN {X 0,Y 573.252,Z 235.292,A -85,B 0,C 180,E1 -2033.842,E2 -2033.842} C_VEL
LIN {X 0,Y 573.343,Z 225.951,A -85,B 0,C 180,E1 -2034.714,E2 -2034.714} C_VEL
LIN {X 0,Y 573.427,Z 215.436,A -85,B 0,C 180,E1 -2035.513,E2 -2035.513} C_VEL
LIN {X 0,Y 573.499,Z 204.311,A -85,B 0,C 180,E1 -2036.191,E2 -2036.191} C_VEL
LIN {X 0,Y 573.641,Z 192.377,A -85,B 0,C 180,E1 -2036.752,E2 -2036.752} C_VEL
LIN {X 0,Y 573.792,Z 178.709,A -85,B 0,C 180,E1 -2037.22,E2 -2037.22} C_VEL
LIN {X 0,Y 573.625,Z 171.896,A -85,B 0,C 180,E1 -2037.395,E2 -2037.395} C_VEL
LIN {X 0,Y 572.961,Z 167.675,A -85,B 0,C 180,E1 -2037.504,E2 -2037.504} C_VEL
LIN {X 0,Y 572.943,Z 164.617,A -85,B 0,C 180,E1 -2039.806,E2 -2039.806} C_VEL
LIN {X 0,Y 572.961,Z 161.446,A -85,B 0,C 180,E1 -2042.218,E2 -2042.218} C_VEL
LIN {X 0,Y 572.968,Z 158.46,A -85,B 0,C 180,E1 -2044.576,E2 -2044.576} C_VEL
LIN {X 0,Y 572.972,Z 155.756,A -85,B 0,C 180,E1 -2046.916,E2 -2046.916} C_VEL
LIN {X 0,Y 573.036,Z 153.159,A -85,B 0,C 180,E1 -2049.165,E2 -2049.165} C_VEL
LIN {X 0,Y 573.014,Z 150.423,A -85,B 0,C 180,E1 -2051.404,E2 -2051.404} C_VEL
LIN {X 0,Y 573.081,Z 147.843,A -85,B 0,C 180,E1 -2053.617,E2 -2053.617} C_VEL
LIN {X 0,Y 573.128,Z 145.216,A -85,B 0,C 180,E1 -2055.803,E2 -2055.803} C_VEL
LIN {X 0,Y 573.148,Z 141.634,A -85,B 0,C 180,E1 -2058.801,E2 -2058.801} C_VEL
LIN {X 0,Y 573.144,Z 141.096,A -85,B 0,C 180,E1 -2059.401,E2 -2059.401} C_VEL
LIN {X 0,Y 573.277,Z 141.076,A -85,B 0,C 180,E1 -2062.25,E2 -2062.25} C_VEL
LIN {X 0,Y 573.304,Z 141.076,A -85,B 0,C 180,E1 -2065.077,E2 -2065.077} C_VEL
LIN {X 0,Y 573.314,Z 141.072,A -85,B 0,C 180,E1 -2067.892,E2 -2067.892} C_VEL
LIN {X 0,Y 573.325,Z 141.07,A -85,B 0,C 180,E1 -2070.702,E2 -2070.702} C_VEL
LIN {X 0,Y 573.301,Z 141.073,A -85,B 0,C 180,E1 -2072.811,E2 -2072.811} C_VEL
LIN {X 0,Y 573.291,Z 141.075,A -85,B 0,C 180,E1 -2075.628,E2 -2075.628} C_VEL
LIN {X 0,Y 573.282,Z 141.078,A -85,B 0,C 180,E1 -2078.459,E2 -2078.459} C_VEL
LIN {X 0,Y 573.269,Z 141.077,A -85,B 0,C 180,E1 -2081.312,E2 -2081.312} C_VEL
LIN {X 0,Y 573.279,Z 141.079,A -85,B 0,C 180,E1 -2084.425,E2 -2084.425} C_VEL
LIN {X 0,Y 573.257,Z 141.08,A -85,B 0,C 180,E1 -2087.112,E2 -2087.112} C_VEL
LIN {X 0,Y 573.252,Z 141.08,A -85,B 0,C 180,E1 -2090.077,E2 -2090.077} C_VEL
LIN {X 0,Y 573.231,Z 141.084,A -85,B 0,C 180,E1 -2093.1,E2 -2093.1} C_VEL
LIN {X 0,Y 573.25,Z 141.082,A -85,B 0,C 180,E1 -2095.41,E2 -2095.41} C_VEL
LIN {X 0,Y 573.249,Z 141.08,A -85,B 0,C 180,E1 -2098.029,E2 -2098.029} C_VEL
LIN {X 0,Y 573.25,Z 141.082,A -85,B 0,C 180,E1 -2100.176,E2 -2100.176} C_VEL
LIN {X 0,Y 573.252,Z 141.082,A -85,B 0,C 180,E1 -2102.645,E2 -2102.645} C_VEL
LIN {X 0,Y 573.205,Z 141.087,A -85,B 0,C 180,E1 -2105.188,E2 -2105.188} C_VEL
LIN {X 0,Y 573.232,Z 141.082,A -85,B 0,C 180,E1 -2107.808,E2 -2107.808} C_VEL
LIN {X 0,Y 573.268,Z 141.077,A -85,B 0,C 180,E1 -2110.528,E2 -2110.528} C_VEL
LIN {X 0,Y 573.243,Z 141.081,A -85,B 0,C 180,E1 -2113.669,E2 -2113.669} C_VEL
LIN {X 0,Y 573.237,Z 141.081,A -85,B 0,C 180,E1 -2116.641,E2 -2116.641} C_VEL
LIN {X 0,Y 573.243,Z 141.083,A -85,B 0,C 180,E1 -2119.475,E2 -2119.475} C_VEL
LIN {X 0,Y 573.236,Z 141.082,A -85,B 0,C 180,E1 -2122.193,E2 -2122.193} C_VEL
LIN {X 0,Y 573.241,Z 141.082,A -85,B 0,C 180,E1 -2125.228,E2 -2125.228} C_VEL
LIN {X 0,Y 573.246,Z 141.081,A -85,B 0,C 180,E1 -2128.185,E2 -2128.185} C_VEL
LIN {X 0,Y 573.261,Z 141.079,A -85,B 0,C 180,E1 -2130.634,E2 -2130.634} C_VEL
LIN {X 0,Y 573.25,Z 141.08,A -85,B 0,C 180,E1 -2133.024,E2 -2133.024} C_VEL
LIN {X 0,Y 573.274,Z 141.078,A -85,B 0,C 180,E1 -2135.366,E2 -2135.366} C_VEL
LIN {X 0,Y 573.231,Z 141.082,A -85,B 0,C 180,E1 -2138.42,E2 -2138.42} C_VEL
LIN {X 0,Y 573.28,Z 141.076,A -85,B 0,C 180,E1 -2140.729,E2 -2140.729} C_VEL
LIN {X 0,Y 573.247,Z 141.083,A -85,B 0,C 180,E1 -2143.622,E2 -2143.622} C_VEL
LIN {X 0,Y 573.231,Z 141.082,A -85,B 0,C 180,E1 -2146.53,E2 -2146.53} C_VEL
LIN {X 0,Y 573.265,Z 141.078,A -85,B 0,C 180,E1 -2148.745,E2 -2148.745} C_VEL
LIN {X 0,Y 573.257,Z 141.078,A -85,B 0,C 180,E1 -2151.54,E2 -2151.54} C_VEL
LIN {X 0,Y 573.251,Z 141.08,A -85,B 0,C 180,E1 -2153.666,E2 -2153.666} C_VEL
LIN {X 0,Y 573.23,Z 141.085,A -85,B 0,C 180,E1 -2155.782,E2 -2155.782} C_VEL
LIN {X 0,Y 573.314,Z 141.073,A -85,B 0,C 180,E1 -2157.893,E2 -2157.893} C_VEL
LIN {X 0,Y 573.332,Z 141.07,A -85,B 0,C 180,E1 -2160.703,E2 -2160.703} C_VEL
LIN {X 0,Y 573.305,Z 141.075,A -85,B 0,C 180,E1 -2162.811,E2 -2162.811} C_VEL
LIN {X 0,Y 573.296,Z 141.075,A -85,B 0,C 180,E1 -2165.628,E2 -2165.628} C_VEL
LIN {X 0,Y 573.257,Z 141.079,A -85,B 0,C 180,E1 -2168.46,E2 -2168.46} C_VEL
LIN {X 0,Y 573.275,Z 141.079,A -85,B 0,C 180,E1 -2171.312,E2 -2171.312} C_VEL
LIN {X 0,Y 573.261,Z 141.078,A -85,B 0,C 180,E1 -2174.194,E2 -2174.194} C_VEL
LIN {X 0,Y 573.261,Z 141.079,A -85,B 0,C 180,E1 -2177.112,E2 -2177.112} C_VEL
LIN {X 0,Y 573.242,Z 141.081,A -85,B 0,C 180,E1 -2180.077,E2 -2180.077} C_VEL
LIN {X 0,Y 573.237,Z 141.084,A -85,B 0,C 180,E1 -2182.338,E2 -2182.338} C_VEL
LIN {X 0,Y 573.258,Z 141.079,A -85,B 0,C 180,E1 -2185.41,E2 -2185.41} C_VEL
LIN {X 0,Y 573.254,Z 141.08,A -85,B 0,C 180,E1 -2188.029,E2 -2188.029} C_VEL
LIN {X 0,Y 573.231,Z 141.084,A -85,B 0,C 180,E1 -2190.882,E2 -2190.882} C_VEL
LIN {X 0,Y 573.243,Z 141.081,A -85,B 0,C 180,E1 -2193.521,E2 -2193.521} C_VEL
LIN {X 0,Y 573.217,Z 141.083,A -85,B 0,C 180,E1 -2196.052,E2 -2196.052} C_VEL
LIN {X 0,Y 573.241,Z 141.081,A -85,B 0,C 180,E1 -2198.702,E2 -2198.702} C_VEL
LIN {X 0,Y 573.231,Z 141.085,A -85,B 0,C 180,E1 -2201.593,E2 -2201.593} C_VEL
LIN {X 0,Y 573.236,Z 141.081,A -85,B 0,C 180,E1 -2204.334,E2 -2204.334} C_VEL
LIN {X 0,Y 573.244,Z 141.081,A -85,B 0,C 180,E1 -2207.359,E2 -2207.359} C_VEL
LIN {X 0,Y 573.253,Z 141.08,A -85,B 0,C 180,E1 -2210.568,E2 -2210.568} C_VEL
LIN {X 0,Y 573.277,Z 141.12,A -85,B 0,C 180,E1 -2213.244,E2 -2213.244} C_VEL
LIN {X 0,Y 573.786,Z 145.917,A -85,B 0,C 180,E1 -2214.853,E2 -2214.853} C_VEL
LIN {X 0,Y 573.666,Z 153.86,A -85,B 0,C 180,E1 -2217.381,E2 -2217.381} C_VEL
LIN {X 0,Y 573.613,Z 162.936,A -85,B 0,C 180,E1 -2220.192,E2 -2220.192} C_VEL
LIN {X 0,Y 573.463,Z 172.395,A -85,B 0,C 180,E1 -2223.035,E2 -2223.035} C_VEL
LIN {X 0,Y 573.393,Z 181.662,A -85,B 0,C 180,E1 -2225.757,E2 -2225.757} C_VEL
LIN {X 0,Y 573.326,Z 190.929,A -85,B 0,C 180,E1 -2228.423,E2 -2228.423} C_VEL
LIN {X 0,Y 573.221,Z 200.33,A -85,B 0,C 180,E1 -2231.078,E2 -2231.078} C_VEL
LIN {X 0,Y 573.161,Z 210.788,A -85,B 0,C 180,E1 -2233.985,E2 -2233.985} C_VEL
LIN {X 0,Y 573.099,Z 221.379,A -85,B 0,C 180,E1 -2236.887,E2 -2236.887} C_VEL
LIN {X 0,Y 573.081,Z 223.53,A -85,B 0,C 180,E1 -2237.472,E2 -2237.472} C_VEL
LIN {X 0,Y 573.864,Z 230.375,A -85,B 0,C 180,E1 -2237.625,E2 -2237.625} C_VEL
LIN {X 0,Y 573.777,Z 242.499,A -85,B 0,C 180,E1 -2237.937,E2 -2237.937} C_VEL
LIN {X 0,Y 573.642,Z 254.529,A -85,B 0,C 180,E1 -2238.383,E2 -2238.383} C_VEL
LIN {X 0,Y 573.51,Z 266.485,A -85,B 0,C 180,E1 -2238.977,E2 -2238.977} C_VEL
LIN {X 0,Y 573.446,Z 277.479,A -85,B 0,C 180,E1 -2239.675,E2 -2239.675} C_VEL
LIN {X 0,Y 573.308,Z 287.648,A -85,B 0,C 180,E1 -2240.474,E2 -2240.474} C_VEL
LIN {X 0,Y 573.215,Z 296.788,A -85,B 0,C 180,E1 -2241.362,E2 -2241.362} C_VEL
LIN {X 0,Y 573.142,Z 305.691,A -85,B 0,C 180,E1 -2242.425,E2 -2242.425} C_VEL
LIN {X 0,Y 573.051,Z 312.407,A -85,B 0,C 180,E1 -2243.415,E2 -2243.415} C_VEL
LIN {X 0,Y 573.07,Z 317.681,A -85,B 0,C 180,E1 -2244.37,E2 -2244.37} C_VEL
LIN {X 0,Y 573.028,Z 322.372,A -85,B 0,C 180,E1 -2245.428,E2 -2245.428} C_VEL
LIN {X 0,Y 573.022,Z 325.957,A -85,B 0,C 180,E1 -2246.484,E2 -2246.484} C_VEL
LIN {X 0,Y 572.959,Z 327.809,A -85,B 0,C 180,E1 -2247.188,E2 -2247.188} C_VEL
LIN {X 0,Y 572.94,Z 329.201,A -85,B 0,C 180,E1 -2247.891,E2 -2247.891} C_VEL
LIN {X 0,Y 572.94,Z 330.784,A -85,B 0,C 180,E1 -2249.297,E2 -2249.297} C_VEL
LIN {X 0,Y 572.938,Z 331,A -85,B 0,C 180,E1 -2250,E2 -2250} C_VEL
LIN {X 0,Y 572.946,Z 330.185,A -85,B 0,C 180,E1 -2251.406,E2 -2251.406} C_VEL
LIN {X 0,Y 572.94,Z 329.201,A -85,B 0,C 180,E1 -2252.109,E2 -2252.109} C_VEL
LIN {X 0,Y 572.959,Z 327.809,A -85,B 0,C 180,E1 -2252.812,E2 -2252.812} C_VEL
LIN {X 0,Y 573.015,Z 324.896,A -85,B 0,C 180,E1 -2253.868,E2 -2253.868} C_VEL
LIN {X 0,Y 572.963,Z 320.949,A -85,B 0,C 180,E1 -2254.926,E2 -2254.926} C_VEL
LIN {X 0,Y 573.065,Z 314.877,A -85,B 0,C 180,E1 -2256.16,E2 -2256.16} C_VEL
LIN {X 0,Y 573.12,Z 308.235,A -85,B 0,C 180,E1 -2257.221,E2 -2257.221} C_VEL
LIN {X 0,Y 573.201,Z 299.988,A -85,B 0,C 180,E1 -2258.283,E2 -2258.283} C_VEL
LIN {X 0,Y 573.287,Z 291.536,A -85,B 0,C 180,E1 -2259.17,E2 -2259.17} C_VEL
LIN {X 0,Y 573.425,Z 281.092,A -85,B 0,C 180,E1 -2260.058,E2 -2260.058} C_VEL
LIN {X 0,Y 573.511,Z 269.535,A -85,B 0,C 180,E1 -2260.847,E2 -2260.847} C_VEL
LIN {X 0,Y 573.611,Z 257.875,A -85,B 0,C 180,E1 -2261.466,E2 -2261.466} C_VEL
LIN {X 0,Y 573.75,Z 245.17,A -85,B 0,C 180,E1 -2261.974,E2 -2261.974} C_VEL
LIN {X 0,Y 573.865,Z 232.515,A -85,B 0,C 180,E1 -2262.331,E2 -2262.331} C_VEL
LIN {X 0,Y 573.571,Z 226.64,A -85,B 0,C 180,E1 -2262.455,E2 -2262.455} C_VEL
LIN {X 0,Y 573.081,Z 223.53,A -85,B 0,C 180,E1 -2262.528,E2 -2262.528} C_VEL
LIN {X 0,Y 573.157,Z 213.435,A -85,B 0,C 180,E1 -2265.286,E2 -2265.286} C_VEL
LIN {X 0,Y 573.214,Z 202.844,A -85,B 0,C 180,E1 -2268.219,E2 -2268.219} C_VEL
LIN {X 0,Y 573.31,Z 193.576,A -85,B 0,C 180,E1 -2270.824,E2 -2270.824} C_VEL
LIN {X 0,Y 573.371,Z 184.31,A -85,B 0,C 180,E1 -2273.476,E2 -2273.476} C_VEL
LIN {X 0,Y 573.455,Z 175.042,A -85,B 0,C 180,E1 -2276.181,E2 -2276.181} C_VEL
LIN {X 0,Y 573.511,Z 165.774,A -85,B 0,C 180,E1 -2278.95,E2 -2278.95} C_VEL
LIN {X 0,Y 573.654,Z 157.831,A -85,B 0,C 180,E1 -2281.378,E2 -2281.378} C_VEL
LIN {X 0,Y 573.773,Z 148.564,A -85,B 0,C 180,E1 -2284.294,E2 -2284.294} C_VEL
LIN {X 0,Y 573.602,Z 143.235,A -85,B 0,C 180,E1 -2286.035,E2 -2286.035} C_VEL
LIN {X 0,Y 573.265,Z 141.081,A -85,B 0,C 180,E1 -2286.812,E2 -2286.812} C_VEL
LIN {X 0,Y 573.244,Z 141.082,A -85,B 0,C 180,E1 -2289.608,E2 -2289.608} C_VEL
LIN {X 0,Y 573.246,Z 141.081,A -85,B 0,C 180,E1 -2292.642,E2 -2292.642} C_VEL
LIN {X 0,Y 573.24,Z 141.082,A -85,B 0,C 180,E1 -2295.667,E2 -2295.667} C_VEL
LIN {X 0,Y 573.234,Z 141.084,A -85,B 0,C 180,E1 -2298.543,E2 -2298.543} C_VEL
LIN {X 0,Y 573.25,Z 141.083,A -85,B 0,C 180,E1 -2301.299,E2 -2301.299} C_VEL
LIN {X 0,Y 573.219,Z 141.085,A -85,B 0,C 180,E1 -2304.018,E2 -2304.018} C_VEL
LIN {X 0,Y 573.291,Z 141.077,A -85,B 0,C 180,E1 -2306.519,E2 -2306.519} C_VEL
LIN {X 0,Y 573.237,Z 141.083,A -85,B 0,C 180,E1 -2309.117,E2 -2309.117} C_VEL
LIN {X 0,Y 573.256,Z 141.08,A -85,B 0,C 180,E1 -2311.971,E2 -2311.971} C_VEL
LIN {X 0,Y 573.259,Z 141.08,A -85,B 0,C 180,E1 -2314.59,E2 -2314.59} C_VEL
LIN {X 0,Y 573.24,Z 141.083,A -85,B 0,C 180,E1 -2317.662,E2 -2317.662} C_VEL
LIN {X 0,Y 573.271,Z 141.079,A -85,B 0,C 180,E1 -2320.67,E2 -2320.67} C_VEL
LIN {X 0,Y 573.248,Z 141.082,A -85,B 0,C 180,E1 -2323.621,E2 -2323.621} C_VEL
LIN {X 0,Y 573.278,Z 141.077,A -85,B 0,C 180,E1 -2325.807,E2 -2325.807} C_VEL
LIN {X 0,Y 573.268,Z 141.079,A -85,B 0,C 180,E1 -2328.745,E2 -2328.745} C_VEL
LIN {X 0,Y 573.289,Z 141.078,A -85,B 0,C 180,E1 -2331.54,E2 -2331.54} C_VEL
LIN {X 0,Y 573.296,Z 141.075,A -85,B 0,C 180,E1 -2334.372,E2 -2334.372} C_VEL
LIN {X 0,Y 573.317,Z 141.073,A -85,B 0,C 180,E1 -2337.892,E2 -2337.892} C_VEL
LIN {X 0,Y 573.338,Z 141.072,A -85,B 0,C 180,E1 -2340.702,E2 -2340.702} C_VEL
LIN {X 0,Y 573.309,Z 141.075,A -85,B 0,C 180,E1 -2342.81,E2 -2342.81} C_VEL
LIN {X 0,Y 573.29,Z 141.078,A -85,B 0,C 180,E1 -2345.628,E2 -2345.628} C_VEL
